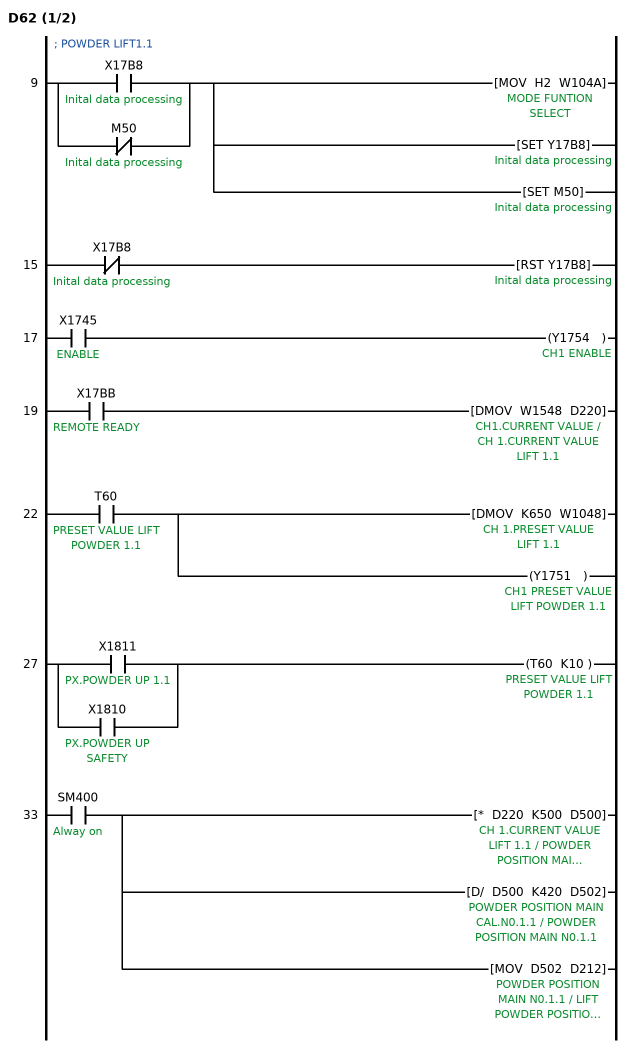
[picture p24: ladder of D62, rungs at steps 9 to 33]
; POWDER LIFT1.1
9     LD      X17B8  ; Inital data processing
      ORI     M50  ; Inital data processing
      MOV     H2 W104A  ; MODE FUNTION SELECT
      SET     Y17B8  ; Inital data processing
      SET     M50  ; Inital data processing
15    LDI     X17B8  ; Inital data processing
      RST     Y17B8  ; Inital data processing
17    LD      X1745  ; ENABLE
      OUT     Y1754  ; CH1 ENABLE
19    LD      X17BB  ; REMOTE READY
      DMOV    W1548 D220  ; CH1.CURRENT VALUE / CH 1.CURRENT VALUE LIFT 1.1
22    LD      T60  ; PRESET VALUE LIFT POWDER 1.1
      DMOV    K650 W1048  ; CH 1.PRESET VALUE LIFT 1.1
      OUT     Y1751  ; CH1 PRESET VALUE LIFT POWDER 1.1
27    LD      X1811  ; PX.POWDER UP 1.1
      OR      X1810  ; PX.POWDER UP SAFETY
      OUT     T60 K10  ; PRESET VALUE LIFT POWDER 1.1
33    LD      SM400  ; Alway on
      *       D220 K500 D500  ; POWDER POSITION MAIN CAL.N0.1.1
      D/      D500 K420 D502  ; POWDER POSITION MAIN N0.1.1
      MOV     D502 D212  ; LIFT POWDER POSITION N0.1.1
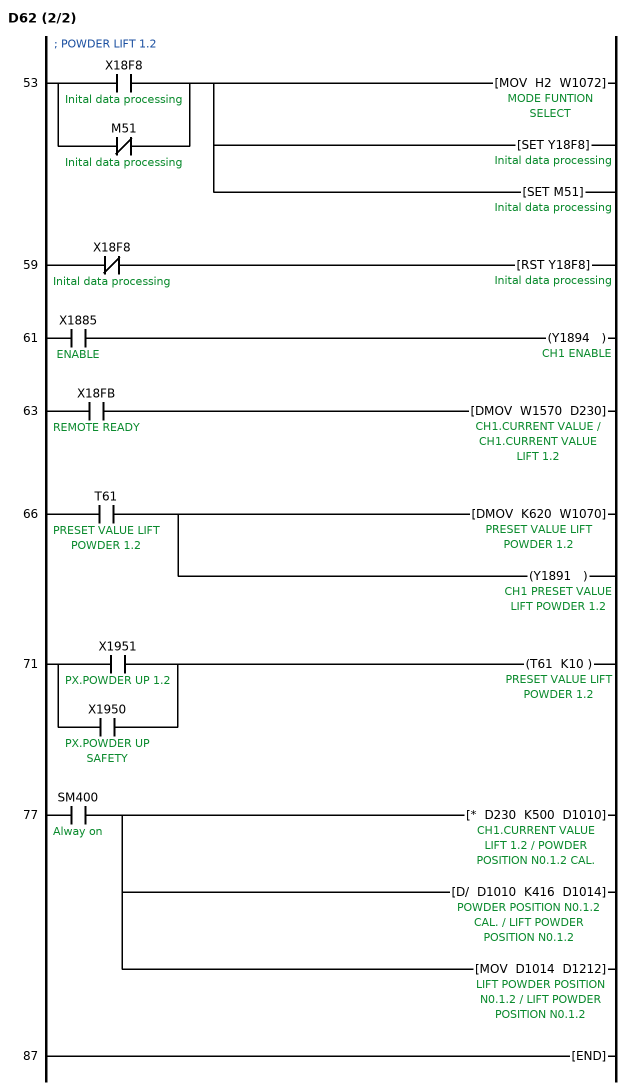
; POWDER LIFT 1.2
53    LD      X18F8  ; Inital data processing
      ORI     M51  ; Inital data processing
      MOV     H2 W1072  ; MODE FUNTION SELECT
      SET     Y18F8  ; Inital data processing
      SET     M51  ; Inital data processing
59    LDI     X18F8  ; Inital data processing
      RST     Y18F8  ; Inital data processing
61    LD      X1885  ; ENABLE
      OUT     Y1894  ; CH1 ENABLE
63    LD      X18FB  ; REMOTE READY
      DMOV    W1570 D230  ; CH1.CURRENT VALUE / CH1.CURRENT VALUE LIFT 1.2
66    LD      T61  ; PRESET VALUE LIFT POWDER 1.2
      DMOV    K620 W1070  ; PRESET VALUE LIFT POWDER 1.2
      OUT     Y1891  ; CH1 PRESET VALUE LIFT POWDER 1.2
71    LD      X1951  ; PX.POWDER UP 1.2
      OR      X1950  ; PX.POWDER UP SAFETY
      OUT     T61 K10  ; PRESET VALUE LIFT POWDER 1.2
77    LD      SM400  ; Alway on
      *       D230 K500 D1010  ; POWDER POSITION N0.1.2 CAL.
      D/      D1010 K416 D1014  ; LIFT POWDER POSITION N0.1.2
      MOV     D1014 D1212  ; LIFT POWDER POSITION N0.1.2
87    END
END_PROGRAM

PROGRAM POWDER1
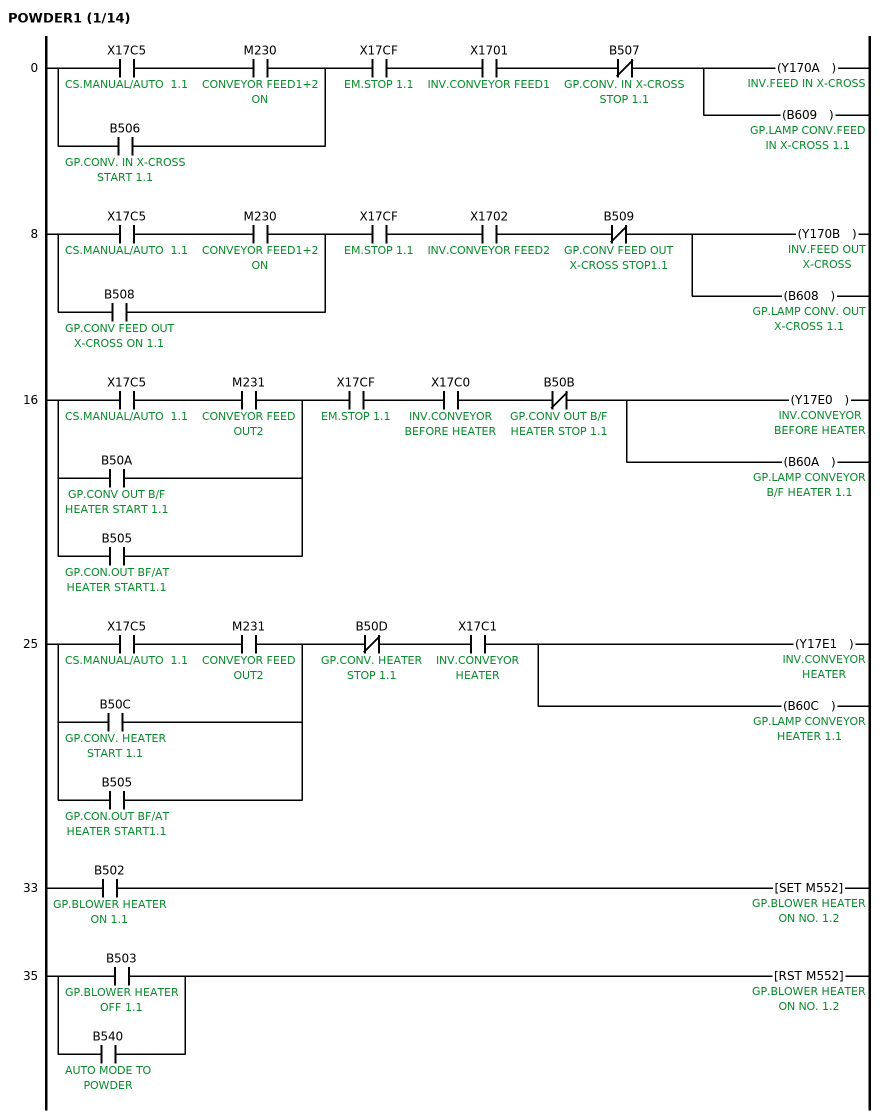
0     LD      X17C5  ; CS.MANUAL/AUTO  1.1
      AND     M230  ; CONVEYOR FEED1+2 ON
      OR      B506  ; GP.CONV. IN X-CROSS START 1.1
      AND     X17CF  ; EM.STOP 1.1
      AND     X1701  ; INV.CONVEYOR FEED1
      ANI     B507  ; GP.CONV. IN X-CROSS STOP 1.1
      OUT     Y170A  ; INV.FEED IN X-CROSS
      OUT     B609  ; GP.LAMP CONV.FEED IN X-CROSS 1.1
8     LD      X17C5  ; CS.MANUAL/AUTO  1.1
      AND     M230  ; CONVEYOR FEED1+2 ON
      OR      B508  ; GP.CONV FEED OUT X-CROSS ON 1.1
      AND     X17CF  ; EM.STOP 1.1
      AND     X1702  ; INV.CONVEYOR FEED2
      ANI     B509  ; GP.CONV FEED OUT X-CROSS STOP1.1
      OUT     Y170B  ; INV.FEED OUT X-CROSS
      OUT     B608  ; GP.LAMP CONV. OUT X-CROSS 1.1
16    LD      X17C5  ; CS.MANUAL/AUTO  1.1
      AND     M231  ; CONVEYOR FEED OUT2
      OR      B50A  ; GP.CONV OUT B/F HEATER START 1.1
      OR      B505  ; GP.CON.OUT BF/AT HEATER START1.1
      AND     X17CF  ; EM.STOP 1.1
      AND     X17C0  ; INV.CONVEYOR BEFORE HEATER
      ANI     B50B  ; GP.CONV OUT B/F HEATER STOP 1.1
      OUT     Y17E0  ; INV.CONVEYOR BEFORE HEATER
      OUT     B60A  ; GP.LAMP CONVEYOR B/F HEATER 1.1
25    LD      X17C5  ; CS.MANUAL/AUTO  1.1
      AND     M231  ; CONVEYOR FEED OUT2
      OR      B50C  ; GP.CONV. HEATER START 1.1
      OR      B505  ; GP.CON.OUT BF/AT HEATER START1.1
      ANI     B50D  ; GP.CONV. HEATER STOP 1.1
      AND     X17C1  ; INV.CONVEYOR HEATER
      OUT     Y17E1  ; INV.CONVEYOR HEATER
      OUT     B60C  ; GP.LAMP CONVEYOR HEATER 1.1
33    LD      B502  ; GP.BLOWER HEATER ON 1.1
      SET     M552  ; GP.BLOWER HEATER ON NO. 1.2
35    LD      B503  ; GP.BLOWER HEATER OFF 1.1
      OR      B540  ; AUTO MODE TO POWDER
      RST     M552  ; GP.BLOWER HEATER ON NO. 1.2
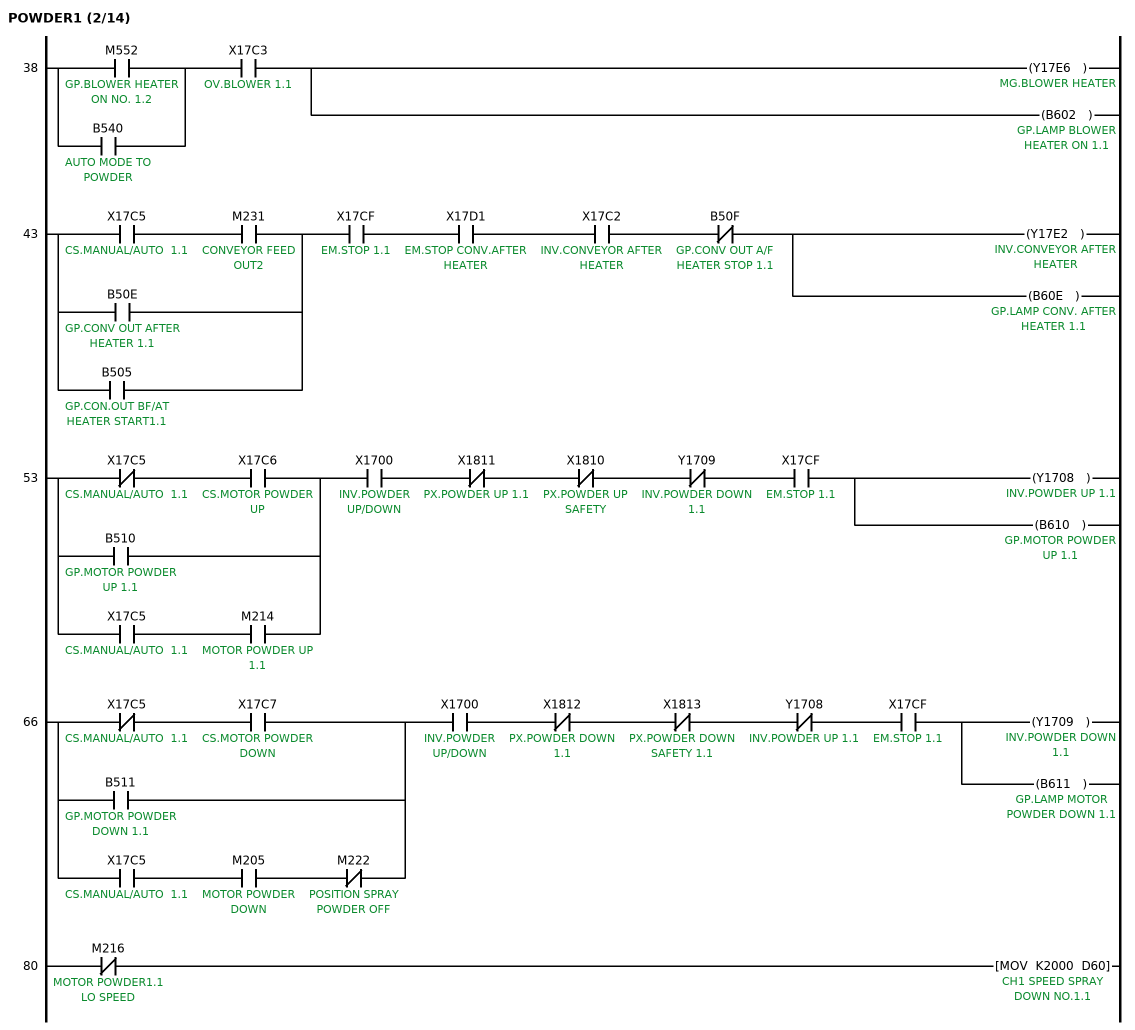
38    LD      M552  ; GP.BLOWER HEATER ON NO. 1.2
      OR      B540  ; AUTO MODE TO POWDER
      AND     X17C3  ; OV.BLOWER 1.1
      OUT     Y17E6  ; MG.BLOWER HEATER
      OUT     B602  ; GP.LAMP BLOWER HEATER ON 1.1
43    LD      X17C5  ; CS.MANUAL/AUTO  1.1
      AND     M231  ; CONVEYOR FEED OUT2
      OR      B50E  ; GP.CONV OUT AFTER HEATER 1.1
      OR      B505  ; GP.CON.OUT BF/AT HEATER START1.1
      AND     X17CF  ; EM.STOP 1.1
      AND     X17D1  ; EM.STOP CONV.AFTER HEATER
      AND     X17C2  ; INV.CONVEYOR AFTER HEATER
      ANI     B50F  ; GP.CONV OUT A/F HEATER STOP 1.1
      OUT     Y17E2  ; INV.CONVEYOR AFTER HEATER
      OUT     B60E  ; GP.LAMP CONV. AFTER HEATER 1.1
53    LDI     X17C5  ; CS.MANUAL/AUTO  1.1
      AND     X17C6  ; CS.MOTOR POWDER UP
      OR      B510  ; GP.MOTOR POWDER UP 1.1
      LD      X17C5  ; CS.MANUAL/AUTO  1.1
      AND     M214  ; MOTOR POWDER UP 1.1
      ORB
      AND     X1700  ; INV.POWDER UP/DOWN
      ANI     X1811  ; PX.POWDER UP 1.1
      ANI     X1810  ; PX.POWDER UP SAFETY
      ANI     Y1709  ; INV.POWDER DOWN 1.1
      AND     X17CF  ; EM.STOP 1.1
      OUT     Y1708  ; INV.POWDER UP 1.1
      OUT     B610  ; GP.MOTOR POWDER UP 1.1
66    LDI     X17C5  ; CS.MANUAL/AUTO  1.1
      AND     X17C7  ; CS.MOTOR POWDER DOWN
      OR      B511  ; GP.MOTOR POWDER DOWN 1.1
      LD      X17C5  ; CS.MANUAL/AUTO  1.1
      AND     M205  ; MOTOR POWDER DOWN
      ANI     M222  ; POSITION SPRAY POWDER OFF
      ORB
      AND     X1700  ; INV.POWDER UP/DOWN
      ANI     X1812  ; PX.POWDER DOWN 1.1
      ANI     X1813  ; PX.POWDER DOWN SAFETY 1.1
      ANI     Y1708  ; INV.POWDER UP 1.1
      AND     X17CF  ; EM.STOP 1.1
      OUT     Y1709  ; INV.POWDER DOWN 1.1
      OUT     B611  ; GP.LAMP MOTOR POWDER DOWN 1.1
80    LDI     M216  ; MOTOR POWDER1.1  LO SPEED
      MOV     K2000 D60  ; CH1 SPEED SPRAY DOWN NO.1.1
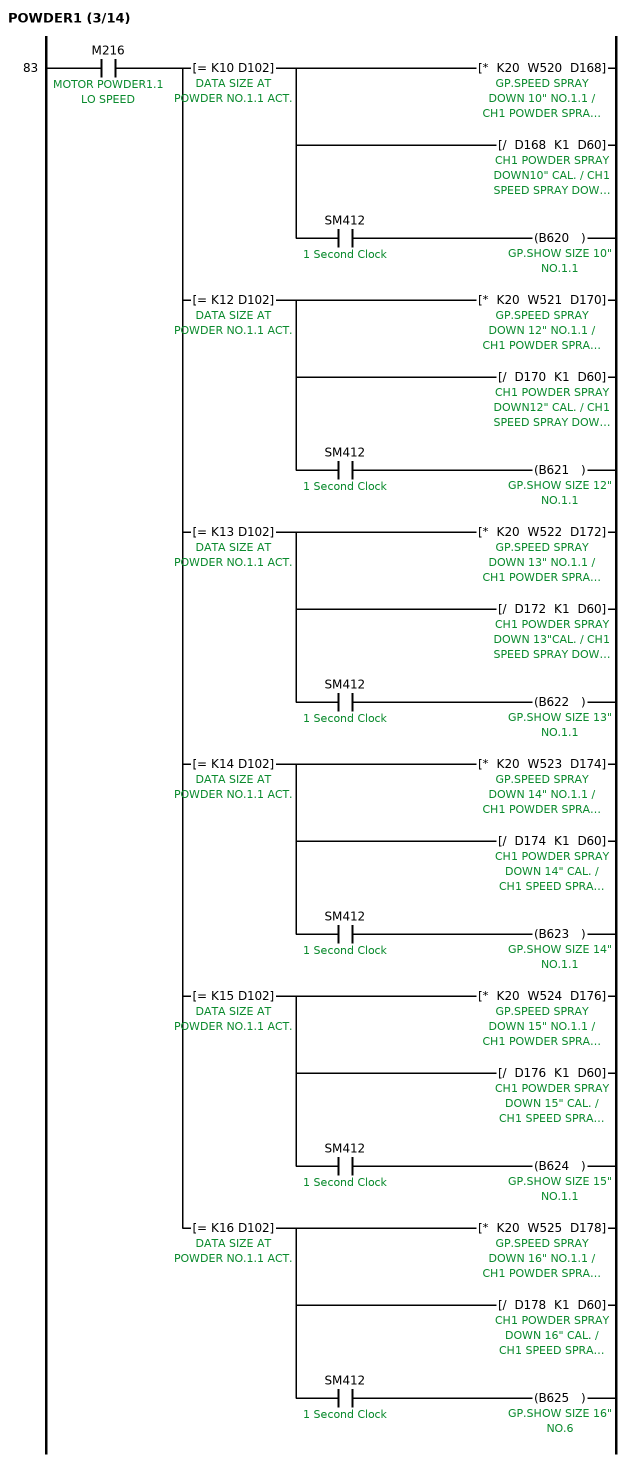
83    LD      M216  ; MOTOR POWDER1.1  LO SPEED
      MPS
      AND=    K10 D102  ; DATA SIZE AT POWDER NO.1.1 ACT.
      *       K20 W520 D168  ; GP.SPEED SPRAY DOWN 10" NO.1.1 / CH1 POWDER SPRAY DOWN10" CAL.
      /       D168 K1 D60
      AND     SM412  ; 1 Second Clock
      OUT     B620  ; GP.SHOW SIZE 10" NO.1.1
      MRD
      AND=    K12 D102  ; DATA SIZE AT POWDER NO.1.1 ACT.
      *       K20 W521 D170  ; GP.SPEED SPRAY DOWN 12" NO.1.1 / CH1 POWDER SPRAY DOWN12" CAL.
      /       D170 K1 D60
      AND     SM412  ; 1 Second Clock
      OUT     B621  ; GP.SHOW SIZE 12" NO.1.1
      MRD
      AND=    K13 D102  ; DATA SIZE AT POWDER NO.1.1 ACT.
      *       K20 W522 D172  ; GP.SPEED SPRAY DOWN 13" NO.1.1 / CH1 POWDER SPRAY DOWN 13"CAL.
      /       D172 K1 D60
      AND     SM412  ; 1 Second Clock
      OUT     B622  ; GP.SHOW SIZE 13" NO.1.1
      MRD
      AND=    K14 D102  ; DATA SIZE AT POWDER NO.1.1 ACT.
      *       K20 W523 D174  ; GP.SPEED SPRAY DOWN 14" NO.1.1 / CH1 POWDER SPRAY DOWN 14" CAL.
      /       D174 K1 D60
      AND     SM412  ; 1 Second Clock
      OUT     B623  ; GP.SHOW SIZE 14" NO.1.1
      MRD
      AND=    K15 D102  ; DATA SIZE AT POWDER NO.1.1 ACT.
      *       K20 W524 D176  ; GP.SPEED SPRAY DOWN 15" NO.1.1 / CH1 POWDER SPRAY DOWN 15" CAL.
      /       D176 K1 D60
      AND     SM412  ; 1 Second Clock
      OUT     B624  ; GP.SHOW SIZE 15" NO.1.1
      MPP
      AND=    K16 D102  ; DATA SIZE AT POWDER NO.1.1 ACT.
      *       K20 W525 D178  ; GP.SPEED SPRAY DOWN 16" NO.1.1 / CH1 POWDER SPRAY DOWN 16" CAL.
      /       D178 K1 D60
      AND     SM412  ; 1 Second Clock
      OUT     B625  ; GP.SHOW SIZE 16" NO.6
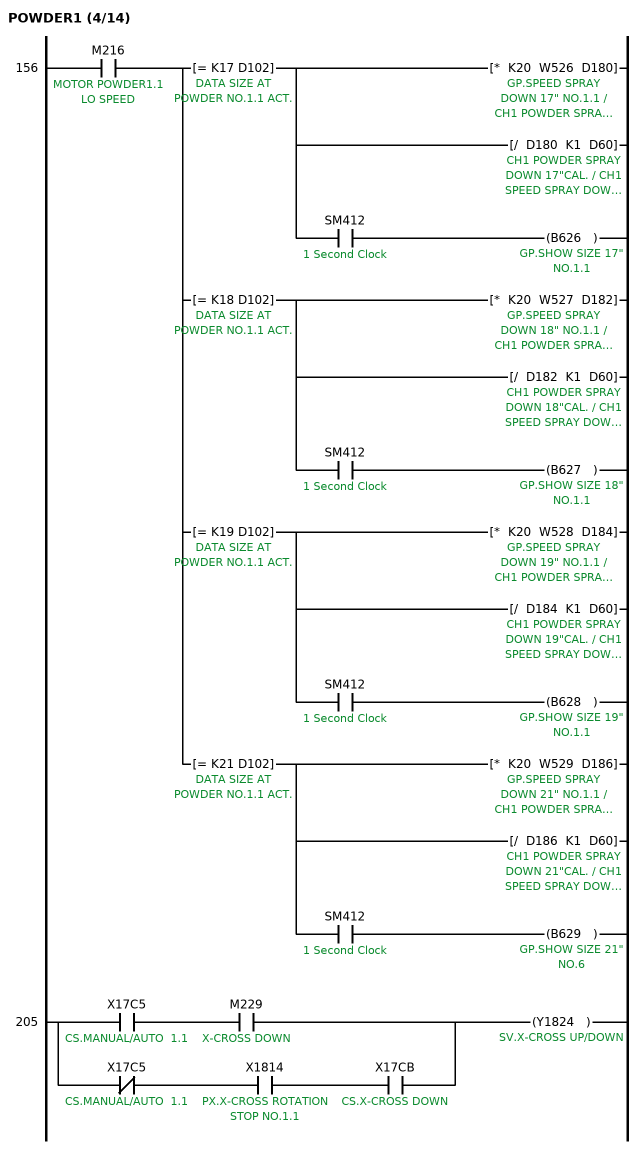
156   LD      M216  ; MOTOR POWDER1.1  LO SPEED
      MPS
      AND=    K17 D102  ; DATA SIZE AT POWDER NO.1.1 ACT.
      *       K20 W526 D180  ; GP.SPEED SPRAY DOWN 17" NO.1.1 / CH1 POWDER SPRAY DOWN 17"CAL.
      /       D180 K1 D60
      AND     SM412  ; 1 Second Clock
      OUT     B626  ; GP.SHOW SIZE 17" NO.1.1
      MRD
      AND=    K18 D102  ; DATA SIZE AT POWDER NO.1.1 ACT.
      *       K20 W527 D182  ; GP.SPEED SPRAY DOWN 18" NO.1.1 / CH1 POWDER SPRAY DOWN 18"CAL.
      /       D182 K1 D60
      AND     SM412  ; 1 Second Clock
      OUT     B627  ; GP.SHOW SIZE 18" NO.1.1
      MRD
      AND=    K19 D102  ; DATA SIZE AT POWDER NO.1.1 ACT.
      *       K20 W528 D184  ; GP.SPEED SPRAY DOWN 19" NO.1.1 / CH1 POWDER SPRAY DOWN 19"CAL.
      /       D184 K1 D60
      AND     SM412  ; 1 Second Clock
      OUT     B628  ; GP.SHOW SIZE 19" NO.1.1
      MPP
      AND=    K21 D102  ; DATA SIZE AT POWDER NO.1.1 ACT.
      *       K20 W529 D186  ; GP.SPEED SPRAY DOWN 21" NO.1.1 / CH1 POWDER SPRAY DOWN 21"CAL.
      /       D186 K1 D60
      AND     SM412  ; 1 Second Clock
      OUT     B629  ; GP.SHOW SIZE 21" NO.6
205   LD      X17C5  ; CS.MANUAL/AUTO  1.1
      AND     M229  ; X-CROSS DOWN
      LDI     X17C5  ; CS.MANUAL/AUTO  1.1
      AND     X1814  ; PX.X-CROSS ROTATION STOP NO.1.1
      AND     X17CB  ; CS.X-CROSS DOWN
      ORB
      OUT     Y1824  ; SV.X-CROSS UP/DOWN
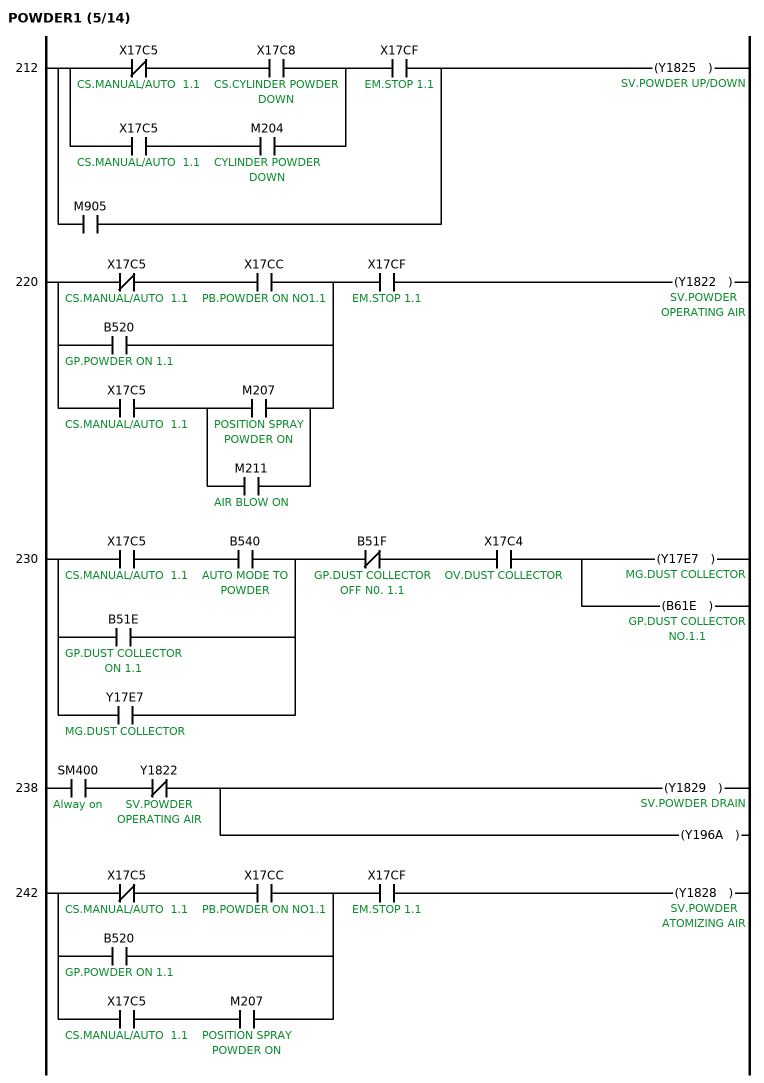
212   LDI     X17C5  ; CS.MANUAL/AUTO  1.1
      AND     X17C8  ; CS.CYLINDER POWDER DOWN
      LD      X17C5  ; CS.MANUAL/AUTO  1.1
      AND     M204  ; CYLINDER POWDER DOWN
      ORB
      AND     X17CF  ; EM.STOP 1.1
      OR      M905
      OUT     Y1825  ; SV.POWDER UP/DOWN
220   LDI     X17C5  ; CS.MANUAL/AUTO  1.1
      AND     X17CC  ; PB.POWDER ON NO1.1
      OR      B520  ; GP.POWDER ON 1.1
      LD      X17C5  ; CS.MANUAL/AUTO  1.1
      LD      M207  ; POSITION SPRAY POWDER ON
      OR      M211  ; AIR BLOW ON
      ANB
      ORB
      AND     X17CF  ; EM.STOP 1.1
      OUT     Y1822  ; SV.POWDER OPERATING AIR
230   LD      X17C5  ; CS.MANUAL/AUTO  1.1
      AND     B540  ; AUTO MODE TO POWDER
      OR      B51E  ; GP.DUST COLLECTOR ON 1.1
      OR      Y17E7  ; MG.DUST COLLECTOR
      ANI     B51F  ; GP.DUST COLLECTOR OFF N0. 1.1
      AND     X17C4  ; OV.DUST COLLECTOR
      OUT     Y17E7  ; MG.DUST COLLECTOR
      OUT     B61E  ; GP.DUST COLLECTOR NO.1.1
238   LD      SM400  ; Alway on
      ANI     Y1822  ; SV.POWDER OPERATING AIR
      OUT     Y1829  ; SV.POWDER DRAIN
      OUT     Y196A
242   LDI     X17C5  ; CS.MANUAL/AUTO  1.1
      AND     X17CC  ; PB.POWDER ON NO1.1
      OR      B520  ; GP.POWDER ON 1.1
      LD      X17C5  ; CS.MANUAL/AUTO  1.1
      AND     M207  ; POSITION SPRAY POWDER ON
      ORB
      AND     X17CF  ; EM.STOP 1.1
      OUT     Y1828  ; SV.POWDER ATOMIZING AIR
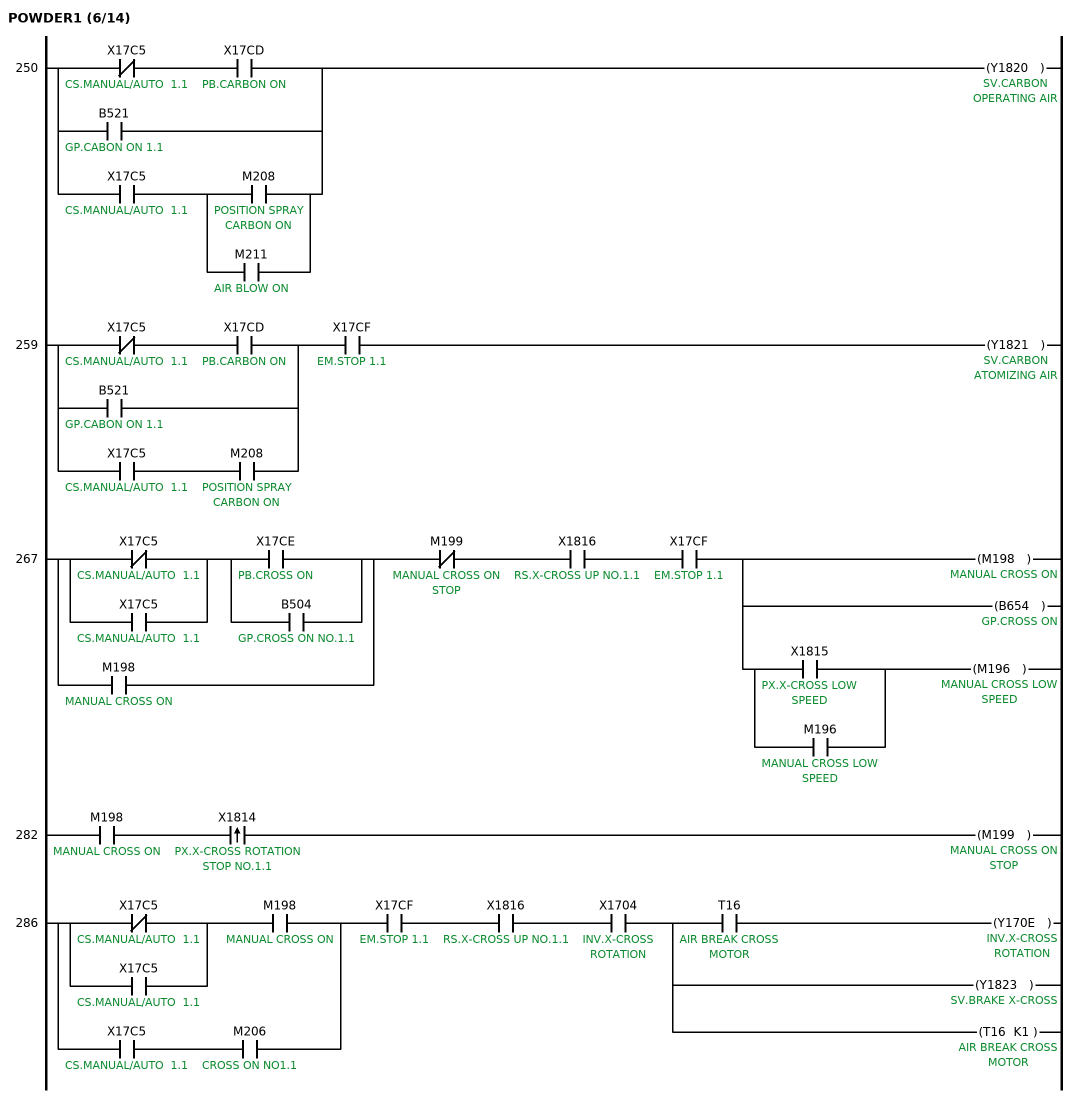
250   LDI     X17C5  ; CS.MANUAL/AUTO  1.1
      AND     X17CD  ; PB.CARBON ON
      OR      B521  ; GP.CABON ON 1.1
      LD      X17C5  ; CS.MANUAL/AUTO  1.1
      LD      M208  ; POSITION SPRAY CARBON ON
      OR      M211  ; AIR BLOW ON
      ANB
      ORB
      OUT     Y1820  ; SV.CARBON OPERATING AIR
259   LDI     X17C5  ; CS.MANUAL/AUTO  1.1
      AND     X17CD  ; PB.CARBON ON
      OR      B521  ; GP.CABON ON 1.1
      LD      X17C5  ; CS.MANUAL/AUTO  1.1
      AND     M208  ; POSITION SPRAY CARBON ON
      ORB
      AND     X17CF  ; EM.STOP 1.1
      OUT     Y1821  ; SV.CARBON ATOMIZING AIR
267   LDI     X17C5  ; CS.MANUAL/AUTO  1.1
      OR      X17C5  ; CS.MANUAL/AUTO  1.1
      LD      X17CE  ; PB.CROSS ON
      OR      B504  ; GP.CROSS ON NO.1.1
      ANB
      OR      M198  ; MANUAL CROSS ON
      ANI     M199  ; MANUAL CROSS ON STOP
      AND     X1816  ; RS.X-CROSS UP NO.1.1
      AND     X17CF  ; EM.STOP 1.1
      OUT     M198  ; MANUAL CROSS ON
      OUT     B654  ; GP.CROSS ON
      LD      X1815  ; PX.X-CROSS LOW SPEED
      OR      M196  ; MANUAL CROSS LOW SPEED
      ANB
      OUT     M196  ; MANUAL CROSS LOW SPEED
282   LD      M198  ; MANUAL CROSS ON
      ANDP    X1814  ; PX.X-CROSS ROTATION STOP NO.1.1
      OUT     M199  ; MANUAL CROSS ON STOP
286   LDI     X17C5  ; CS.MANUAL/AUTO  1.1
      OR      X17C5  ; CS.MANUAL/AUTO  1.1
      AND     M198  ; MANUAL CROSS ON
      LD      X17C5  ; CS.MANUAL/AUTO  1.1
      AND     M206  ; CROSS ON NO1.1
      ORB
      AND     X17CF  ; EM.STOP 1.1
      AND     X1816  ; RS.X-CROSS UP NO.1.1
      AND     X1704  ; INV.X-CROSS ROTATION
      MPS
      AND     T16  ; AIR BREAK CROSS MOTOR
      OUT     Y170E  ; INV.X-CROSS ROTATION
      MPP
      OUT     Y1823  ; SV.BRAKE X-CROSS
      OUT     T16 K1  ; AIR BREAK CROSS MOTOR
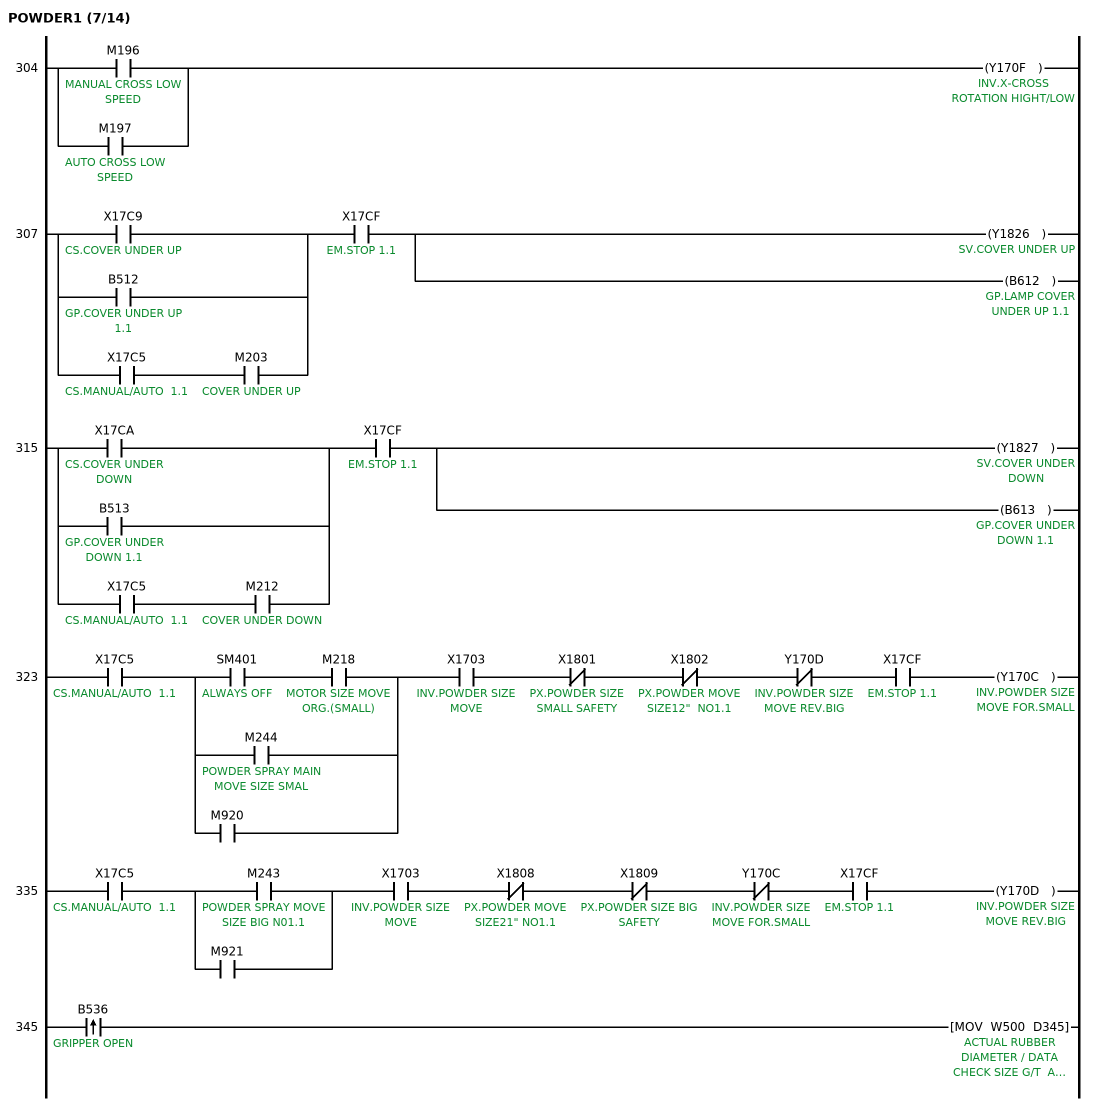
304   LD      M196  ; MANUAL CROSS LOW SPEED
      OR      M197  ; AUTO CROSS LOW SPEED
      OUT     Y170F  ; INV.X-CROSS ROTATION HIGHT/LOW
307   LD      X17C9  ; CS.COVER UNDER UP
      OR      B512  ; GP.COVER UNDER UP 1.1
      LD      X17C5  ; CS.MANUAL/AUTO  1.1
      AND     M203  ; COVER UNDER UP
      ORB
      AND     X17CF  ; EM.STOP 1.1
      OUT     Y1826  ; SV.COVER UNDER UP
      OUT     B612  ; GP.LAMP COVER UNDER UP 1.1
315   LD      X17CA  ; CS.COVER UNDER DOWN
      OR      B513  ; GP.COVER UNDER DOWN 1.1
      LD      X17C5  ; CS.MANUAL/AUTO  1.1
      AND     M212  ; COVER UNDER DOWN
      ORB
      AND     X17CF  ; EM.STOP 1.1
      OUT     Y1827  ; SV.COVER UNDER DOWN
      OUT     B613  ; GP.COVER UNDER DOWN 1.1
323   LD      X17C5  ; CS.MANUAL/AUTO  1.1
      LD      SM401  ; ALWAYS OFF
      AND     M218  ; MOTOR SIZE MOVE ORG.(SMALL)
      OR      M244  ; POWDER SPRAY MAIN MOVE SIZE SMAL
      OR      M920
      ANB
      AND     X1703  ; INV.POWDER SIZE MOVE
      ANI     X1801  ; PX.POWDER SIZE SMALL SAFETY
      ANI     X1802  ; PX.POWDER MOVE  SIZE12"  NO1.1
      ANI     Y170D  ; INV.POWDER SIZE MOVE REV.BIG
      AND     X17CF  ; EM.STOP 1.1
      OUT     Y170C  ; INV.POWDER SIZE MOVE FOR.SMALL
335   LD      X17C5  ; CS.MANUAL/AUTO  1.1
      LD      M243  ; POWDER SPRAY MOVE SIZE BIG N01.1
      OR      M921
      ANB
      AND     X1703  ; INV.POWDER SIZE MOVE
      ANI     X1808  ; PX.POWDER MOVE SIZE21" NO1.1
      ANI     X1809  ; PX.POWDER SIZE BIG SAFETY
      ANI     Y170C  ; INV.POWDER SIZE MOVE FOR.SMALL
      AND     X17CF  ; EM.STOP 1.1
      OUT     Y170D  ; INV.POWDER SIZE MOVE REV.BIG
345   LDP     B536  ; GRIPPER OPEN
      MOV     W500 D345  ; ACTUAL RUBBER DIAMETER / DATA CHECK SIZE G/T  AT ROBOT
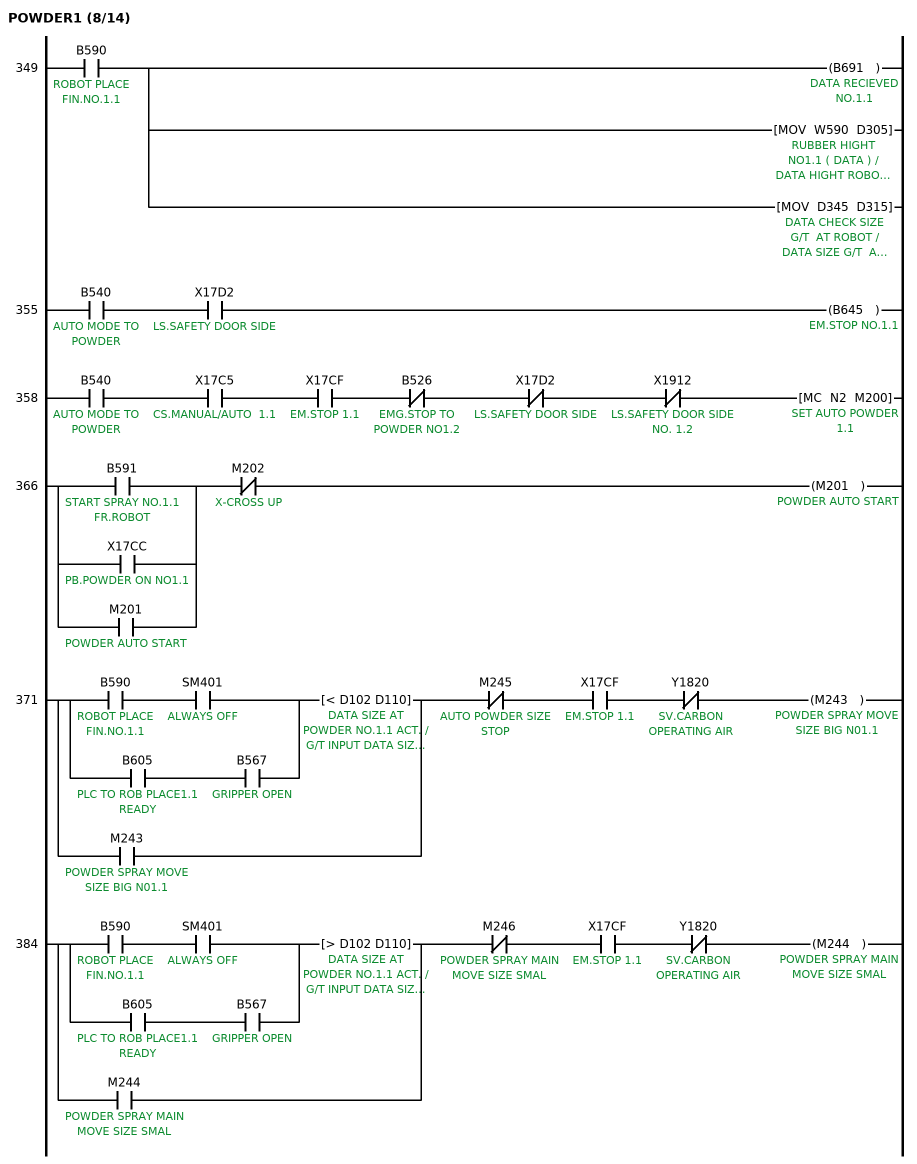
349   LD      B590  ; ROBOT PLACE FIN.NO.1.1
      OUT     B691  ; DATA RECIEVED NO.1.1
      MOV     W590 D305  ; RUBBER HIGHT NO1.1 ( DATA ) / DATA HIGHT ROBOT TO N0.1.1
      MOV     D345 D315  ; DATA SIZE G/T  AT ROBOT NO.1.1
355   LD      B540  ; AUTO MODE TO POWDER
      AND     X17D2  ; LS.SAFETY DOOR SIDE
      OUT     B645  ; EM.STOP NO.1.1
358   LD      B540  ; AUTO MODE TO POWDER
      AND     X17C5  ; CS.MANUAL/AUTO  1.1
      AND     X17CF  ; EM.STOP 1.1
      ANI     B526  ; EMG.STOP TO POWDER NO1.2
      ANI     X17D2  ; LS.SAFETY DOOR SIDE
      ANI     X1912  ; LS.SAFETY DOOR SIDE NO. 1.2
      MC      N2 M200  ; SET AUTO POWDER 1.1
366   LD      B591  ; START SPRAY NO.1.1 FR.ROBOT
      OR      X17CC  ; PB.POWDER ON NO1.1
      OR      M201  ; POWDER AUTO START
      ANI     M202  ; X-CROSS UP
      OUT     M201  ; POWDER AUTO START
371   LD      B590  ; ROBOT PLACE FIN.NO.1.1
      AND     SM401  ; ALWAYS OFF
      LD      B605  ; PLC TO ROB PLACE1.1 READY
      AND     B567  ; GRIPPER OPEN
      ORB
      AND<    D102 D110  ; DATA SIZE AT POWDER NO.1.1 ACT. / G/T INPUT DATA SIZE AT ROBOT
      OR      M243  ; POWDER SPRAY MOVE SIZE BIG N01.1
      ANI     M245  ; AUTO POWDER SIZE STOP
      AND     X17CF  ; EM.STOP 1.1
      ANI     Y1820  ; SV.CARBON OPERATING AIR
      OUT     M243  ; POWDER SPRAY MOVE SIZE BIG N01.1
384   LD      B590  ; ROBOT PLACE FIN.NO.1.1
      AND     SM401  ; ALWAYS OFF
      LD      B605  ; PLC TO ROB PLACE1.1 READY
      AND     B567  ; GRIPPER OPEN
      ORB
      AND>    D102 D110  ; DATA SIZE AT POWDER NO.1.1 ACT. / G/T INPUT DATA SIZE AT ROBOT
      OR      M244  ; POWDER SPRAY MAIN MOVE SIZE SMAL
      ANI     M246  ; POWDER SPRAY MAIN MOVE SIZE SMAL
      AND     X17CF  ; EM.STOP 1.1
      ANI     Y1820  ; SV.CARBON OPERATING AIR
      OUT     M244  ; POWDER SPRAY MAIN MOVE SIZE SMAL
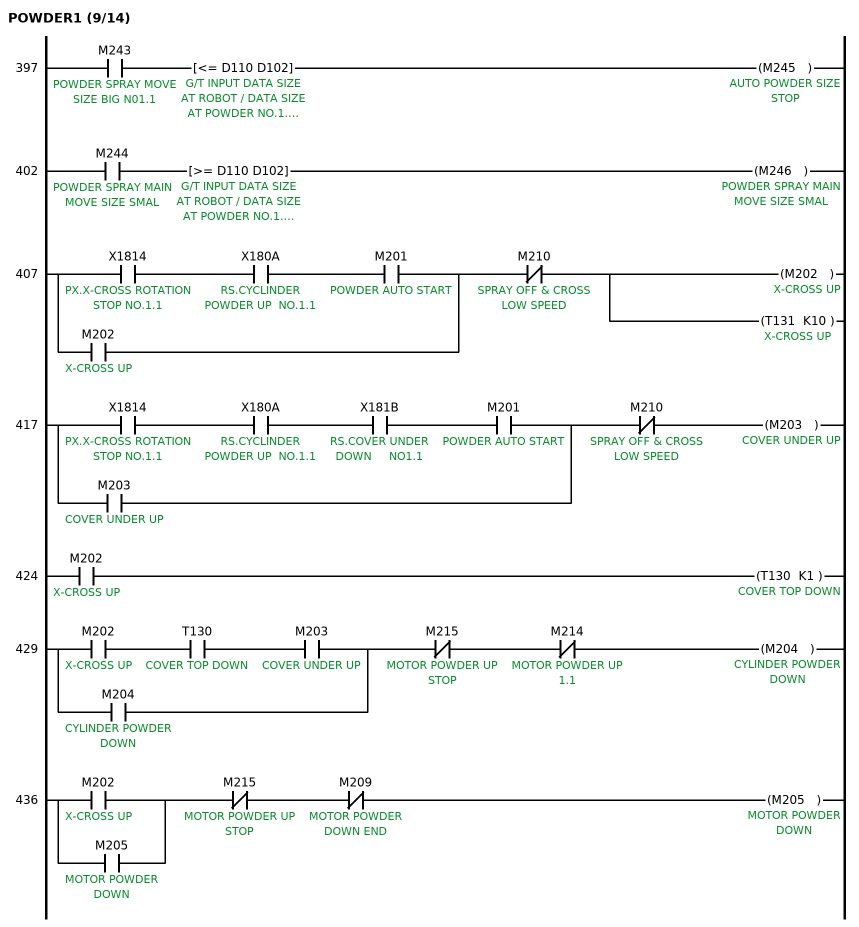
397   LD      M243  ; POWDER SPRAY MOVE SIZE BIG N01.1
      AND<=   D110 D102  ; G/T INPUT DATA SIZE AT ROBOT / DATA SIZE AT POWDER NO.1.1 ACT.
      OUT     M245  ; AUTO POWDER SIZE STOP
402   LD      M244  ; POWDER SPRAY MAIN MOVE SIZE SMAL
      AND>=   D110 D102  ; G/T INPUT DATA SIZE AT ROBOT / DATA SIZE AT POWDER NO.1.1 ACT.
      OUT     M246  ; POWDER SPRAY MAIN MOVE SIZE SMAL
407   LD      X1814  ; PX.X-CROSS ROTATION STOP NO.1.1
      AND     X180A  ; RS.CYCLINDER POWDER UP  NO.1.1
      AND     M201  ; POWDER AUTO START
      OR      M202  ; X-CROSS UP
      ANI     M210  ; SPRAY OFF & CROSS LOW SPEED
      OUT     M202  ; X-CROSS UP
      OUT     T131 K10  ; X-CROSS UP
417   LD      X1814  ; PX.X-CROSS ROTATION STOP NO.1.1
      AND     X180A  ; RS.CYCLINDER POWDER UP  NO.1.1
      AND     X181B  ; RS.COVER UNDER DOWN     NO1.1
      AND     M201  ; POWDER AUTO START
      OR      M203  ; COVER UNDER UP
      ANI     M210  ; SPRAY OFF & CROSS LOW SPEED
      OUT     M203  ; COVER UNDER UP
424   LD      M202  ; X-CROSS UP
      OUT     T130 K1  ; COVER TOP DOWN
429   LD      M202  ; X-CROSS UP
      AND     T130  ; COVER TOP DOWN
      AND     M203  ; COVER UNDER UP
      OR      M204  ; CYLINDER POWDER DOWN
      ANI     M215  ; MOTOR POWDER UP STOP
      ANI     M214  ; MOTOR POWDER UP 1.1
      OUT     M204  ; CYLINDER POWDER DOWN
436   LD      M202  ; X-CROSS UP
      OR      M205  ; MOTOR POWDER DOWN
      ANI     M215  ; MOTOR POWDER UP STOP
      ANI     M209  ; MOTOR POWDER DOWN END
      OUT     M205  ; MOTOR POWDER DOWN
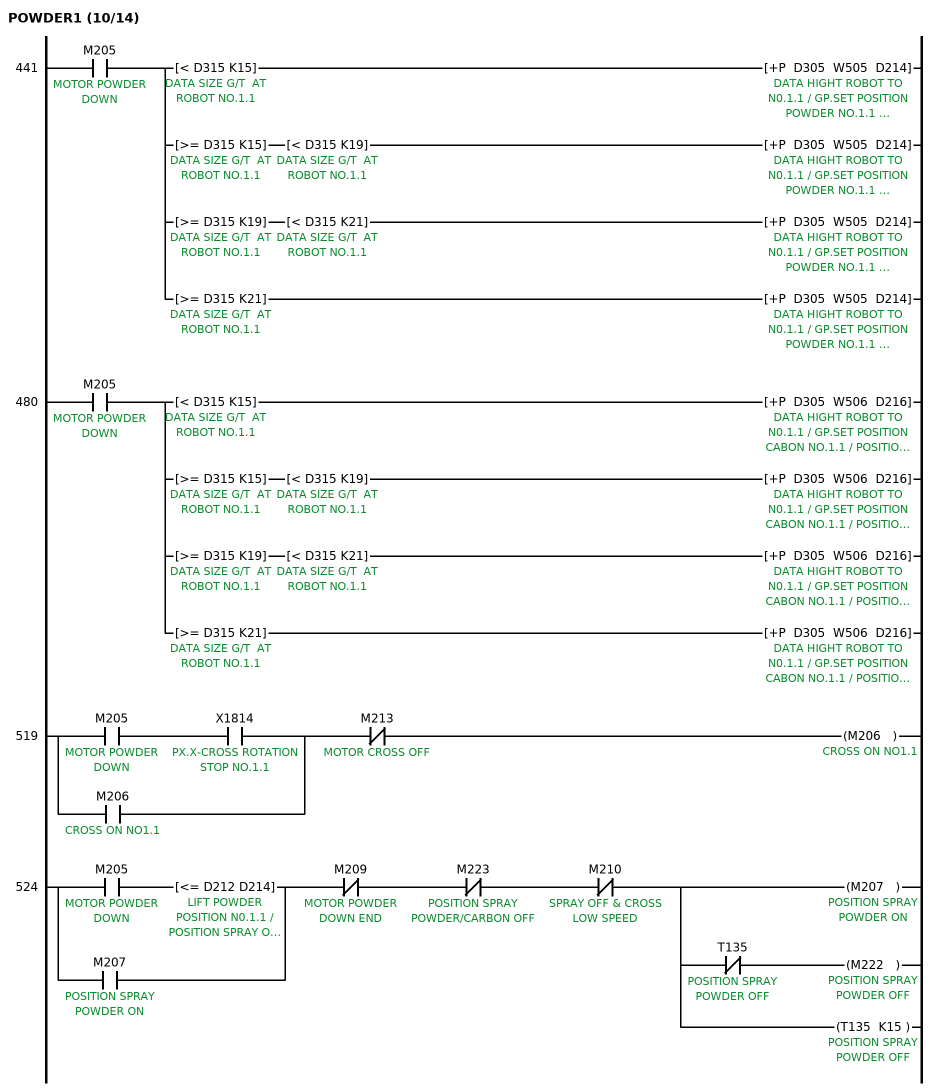
441   LD      M205  ; MOTOR POWDER DOWN
      MPS
      AND<    D315 K15  ; DATA SIZE G/T  AT ROBOT NO.1.1
      +P      D305 W505 D214  ; GP.SET POSITION POWDER NO.1.1 / POSITION SPRAY ON 1.1
      MRD
      AND>=   D315 K15  ; DATA SIZE G/T  AT ROBOT NO.1.1
      AND<    D315 K19  ; DATA SIZE G/T  AT ROBOT NO.1.1
      +P      D305 W505 D214
      MRD
      AND>=   D315 K19  ; DATA SIZE G/T  AT ROBOT NO.1.1
      AND<    D315 K21  ; DATA SIZE G/T  AT ROBOT NO.1.1
      +P      D305 W505 D214
      MPP
      AND>=   D315 K21  ; DATA SIZE G/T  AT ROBOT NO.1.1
      +P      D305 W505 D214
480   LD      M205  ; MOTOR POWDER DOWN
      MPS
      AND<    D315 K15  ; DATA SIZE G/T  AT ROBOT NO.1.1
      +P      D305 W506 D216  ; GP.SET POSITION CABON NO.1.1 / POSITION CARBON ON 1.1
      MRD
      AND>=   D315 K15  ; DATA SIZE G/T  AT ROBOT NO.1.1
      AND<    D315 K19  ; DATA SIZE G/T  AT ROBOT NO.1.1
      +P      D305 W506 D216
      MRD
      AND>=   D315 K19  ; DATA SIZE G/T  AT ROBOT NO.1.1
      AND<    D315 K21  ; DATA SIZE G/T  AT ROBOT NO.1.1
      +P      D305 W506 D216
      MPP
      AND>=   D315 K21  ; DATA SIZE G/T  AT ROBOT NO.1.1
      +P      D305 W506 D216
519   LD      M205  ; MOTOR POWDER DOWN
      AND     X1814  ; PX.X-CROSS ROTATION STOP NO.1.1
      OR      M206  ; CROSS ON NO1.1
      ANI     M213  ; MOTOR CROSS OFF
      OUT     M206  ; CROSS ON NO1.1
524   LD      M205  ; MOTOR POWDER DOWN
      AND<=   D212 D214  ; LIFT POWDER POSITION N0.1.1 / POSITION SPRAY ON 1.1
      OR      M207  ; POSITION SPRAY POWDER ON
      ANI     M209  ; MOTOR POWDER DOWN END
      ANI     M223  ; POSITION SPRAY POWDER/CARBON OFF
      ANI     M210  ; SPRAY OFF & CROSS LOW SPEED
      OUT     M207  ; POSITION SPRAY POWDER ON
      MPS
      ANI     T135  ; POSITION SPRAY POWDER OFF
      OUT     M222  ; POSITION SPRAY POWDER OFF
      MPP
      OUT     T135 K15  ; POSITION SPRAY POWDER OFF
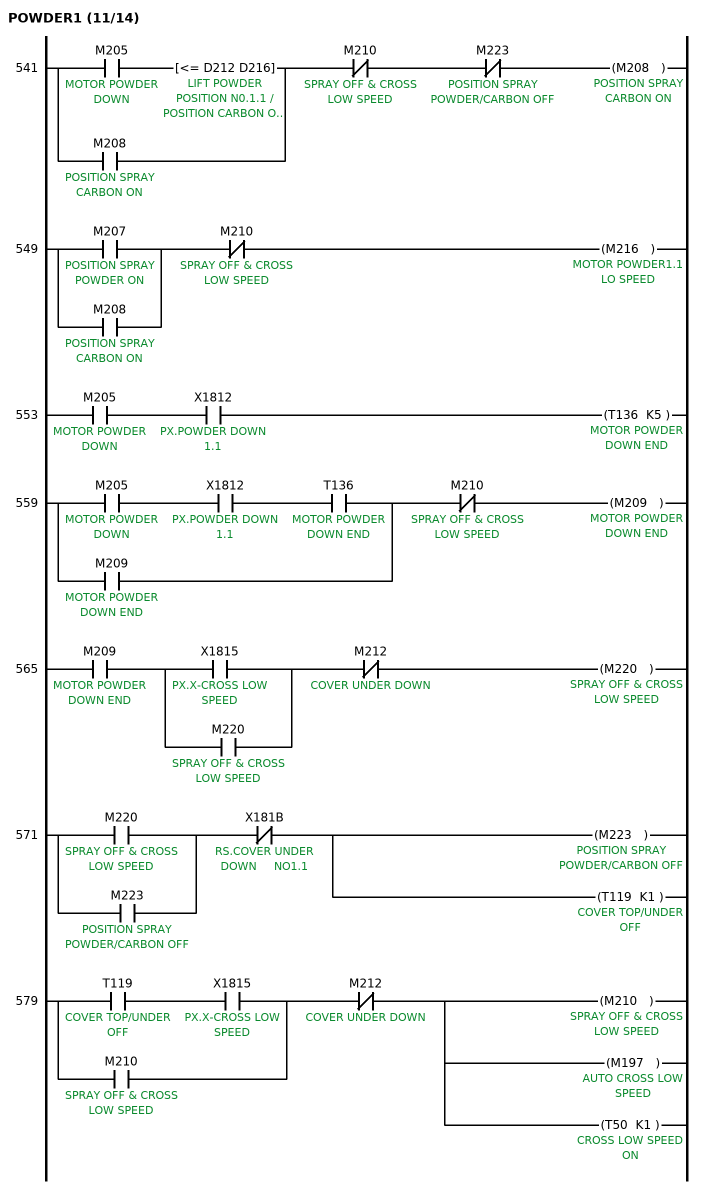
541   LD      M205  ; MOTOR POWDER DOWN
      AND<=   D212 D216  ; LIFT POWDER POSITION N0.1.1 / POSITION CARBON ON 1.1
      OR      M208  ; POSITION SPRAY CARBON ON
      ANI     M210  ; SPRAY OFF & CROSS LOW SPEED
      ANI     M223  ; POSITION SPRAY POWDER/CARBON OFF
      OUT     M208  ; POSITION SPRAY CARBON ON
549   LD      M207  ; POSITION SPRAY POWDER ON
      OR      M208  ; POSITION SPRAY CARBON ON
      ANI     M210  ; SPRAY OFF & CROSS LOW SPEED
      OUT     M216  ; MOTOR POWDER1.1  LO SPEED
553   LD      M205  ; MOTOR POWDER DOWN
      AND     X1812  ; PX.POWDER DOWN 1.1
      OUT     T136 K5  ; MOTOR POWDER DOWN END
559   LD      M205  ; MOTOR POWDER DOWN
      AND     X1812  ; PX.POWDER DOWN 1.1
      AND     T136  ; MOTOR POWDER DOWN END
      OR      M209  ; MOTOR POWDER DOWN END
      ANI     M210  ; SPRAY OFF & CROSS LOW SPEED
      OUT     M209  ; MOTOR POWDER DOWN END
565   LD      M209  ; MOTOR POWDER DOWN END
      LD      X1815  ; PX.X-CROSS LOW SPEED
      OR      M220  ; SPRAY OFF & CROSS LOW SPEED
      ANB
      ANI     M212  ; COVER UNDER DOWN
      OUT     M220  ; SPRAY OFF & CROSS LOW SPEED
571   LD      M220  ; SPRAY OFF & CROSS LOW SPEED
      OR      M223  ; POSITION SPRAY POWDER/CARBON OFF
      ANI     X181B  ; RS.COVER UNDER DOWN     NO1.1
      OUT     M223  ; POSITION SPRAY POWDER/CARBON OFF
      OUT     T119 K1  ; COVER TOP/UNDER OFF
579   LD      T119  ; COVER TOP/UNDER OFF
      AND     X1815  ; PX.X-CROSS LOW SPEED
      OR      M210  ; SPRAY OFF & CROSS LOW SPEED
      ANI     M212  ; COVER UNDER DOWN
      OUT     M210  ; SPRAY OFF & CROSS LOW SPEED
      OUT     M197  ; AUTO CROSS LOW SPEED
      OUT     T50 K1  ; CROSS LOW SPEED ON
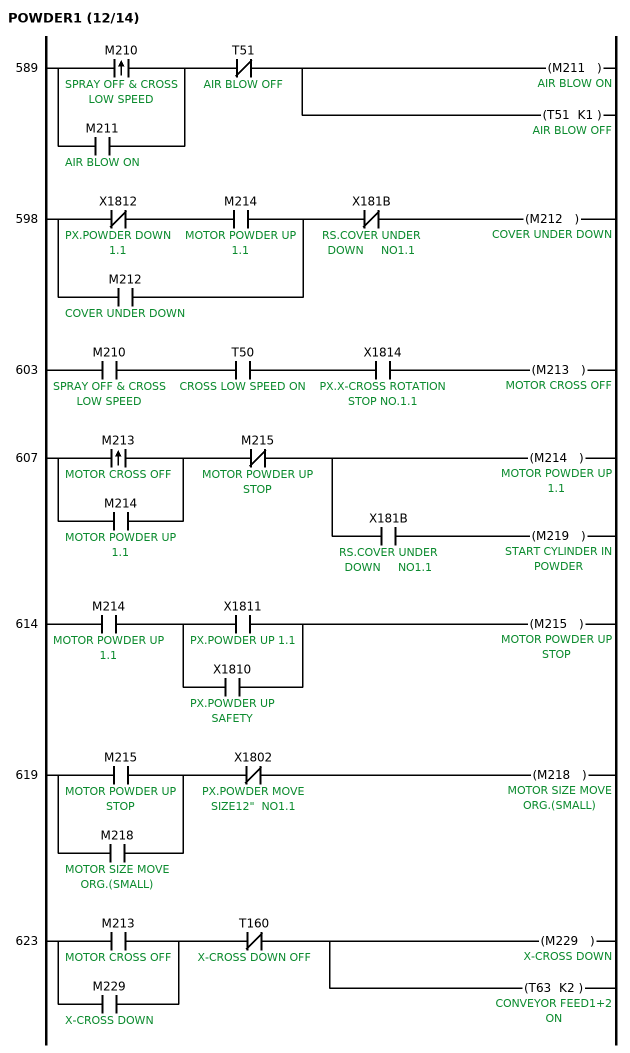
589   LDP     M210  ; SPRAY OFF & CROSS LOW SPEED
      OR      M211  ; AIR BLOW ON
      ANI     T51  ; AIR BLOW OFF
      OUT     M211  ; AIR BLOW ON
      OUT     T51 K1  ; AIR BLOW OFF
598   LDI     X1812  ; PX.POWDER DOWN 1.1
      AND     M214  ; MOTOR POWDER UP 1.1
      OR      M212  ; COVER UNDER DOWN
      ANI     X181B  ; RS.COVER UNDER DOWN     NO1.1
      OUT     M212  ; COVER UNDER DOWN
603   LD      M210  ; SPRAY OFF & CROSS LOW SPEED
      AND     T50  ; CROSS LOW SPEED ON
      AND     X1814  ; PX.X-CROSS ROTATION STOP NO.1.1
      OUT     M213  ; MOTOR CROSS OFF
607   LDP     M213  ; MOTOR CROSS OFF
      OR      M214  ; MOTOR POWDER UP 1.1
      ANI     M215  ; MOTOR POWDER UP STOP
      OUT     M214  ; MOTOR POWDER UP 1.1
      AND     X181B  ; RS.COVER UNDER DOWN     NO1.1
      OUT     M219  ; START CYLINDER IN POWDER
614   LD      M214  ; MOTOR POWDER UP 1.1
      LD      X1811  ; PX.POWDER UP 1.1
      OR      X1810  ; PX.POWDER UP SAFETY
      ANB
      OUT     M215  ; MOTOR POWDER UP STOP
619   LD      M215  ; MOTOR POWDER UP STOP
      OR      M218  ; MOTOR SIZE MOVE ORG.(SMALL)
      ANI     X1802  ; PX.POWDER MOVE  SIZE12"  NO1.1
      OUT     M218  ; MOTOR SIZE MOVE ORG.(SMALL)
623   LD      M213  ; MOTOR CROSS OFF
      OR      M229  ; X-CROSS DOWN
      ANI     T160  ; X-CROSS DOWN OFF
      OUT     M229  ; X-CROSS DOWN
      OUT     T63 K2  ; CONVEYOR FEED1+2 ON
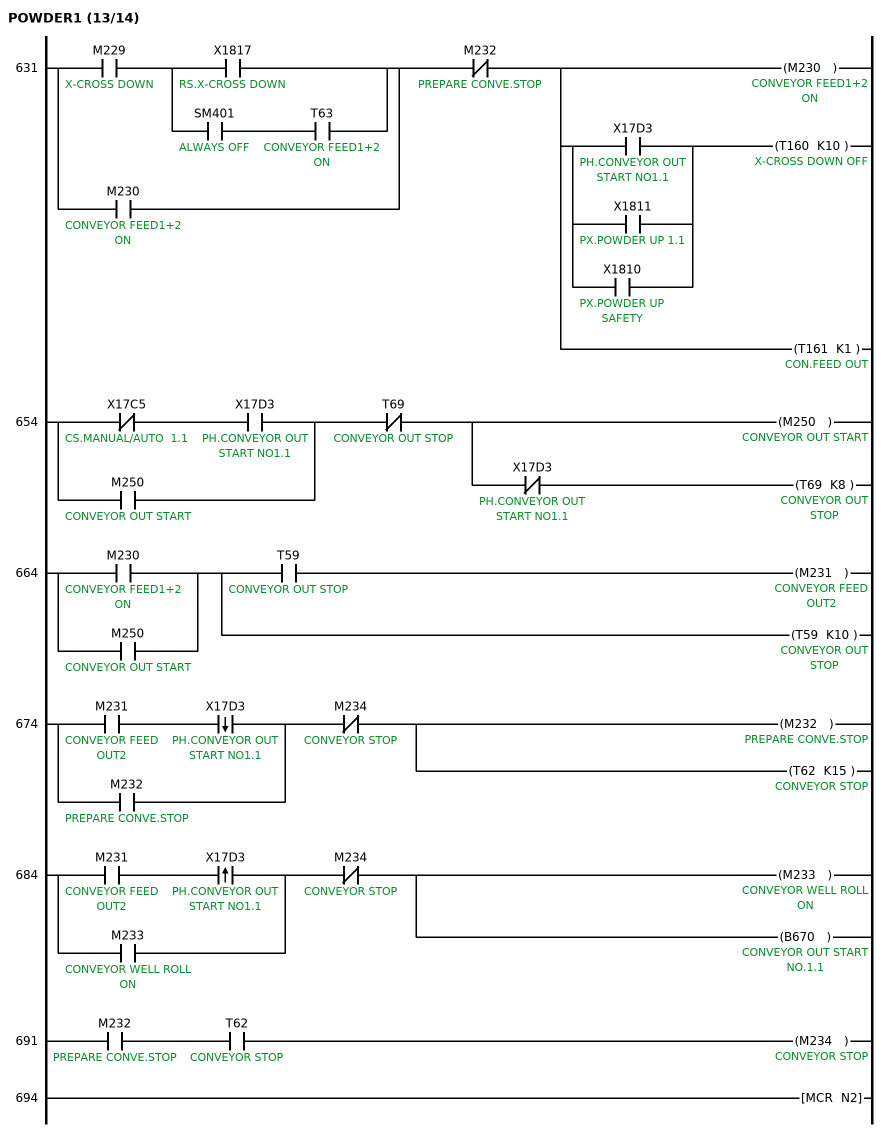
631   LD      M229  ; X-CROSS DOWN
      LD      X1817  ; RS.X-CROSS DOWN
      LD      SM401  ; ALWAYS OFF
      AND     T63  ; CONVEYOR FEED1+2 ON
      ORB
      ANB
      OR      M230  ; CONVEYOR FEED1+2 ON
      ANI     M232  ; PREPARE CONVE.STOP
      OUT     M230  ; CONVEYOR FEED1+2 ON
      MPS
      LD      X17D3  ; PH.CONVEYOR OUT START NO1.1
      OR      X1811  ; PX.POWDER UP 1.1
      OR      X1810  ; PX.POWDER UP SAFETY
      ANB
      OUT     T160 K10  ; X-CROSS DOWN OFF
      MPP
      OUT     T161 K1  ; CON.FEED OUT
654   LDI     X17C5  ; CS.MANUAL/AUTO  1.1
      AND     X17D3  ; PH.CONVEYOR OUT START NO1.1
      OR      M250  ; CONVEYOR OUT START
      ANI     T69  ; CONVEYOR OUT STOP
      OUT     M250  ; CONVEYOR OUT START
      ANI     X17D3  ; PH.CONVEYOR OUT START NO1.1
      OUT     T69 K8  ; CONVEYOR OUT STOP
664   LD      M230  ; CONVEYOR FEED1+2 ON
      OR      M250  ; CONVEYOR OUT START
      MPS
      AND     T59  ; CONVEYOR OUT STOP
      OUT     M231  ; CONVEYOR FEED OUT2
      MPP
      OUT     T59 K10  ; CONVEYOR OUT STOP
674   LD      M231  ; CONVEYOR FEED OUT2
      ANDF    X17D3  ; PH.CONVEYOR OUT START NO1.1
      OR      M232  ; PREPARE CONVE.STOP
      ANI     M234  ; CONVEYOR STOP
      OUT     M232  ; PREPARE CONVE.STOP
      OUT     T62 K15  ; CONVEYOR STOP
684   LD      M231  ; CONVEYOR FEED OUT2
      ANDP    X17D3  ; PH.CONVEYOR OUT START NO1.1
      OR      M233  ; CONVEYOR WELL ROLL ON
      ANI     M234  ; CONVEYOR STOP
      OUT     M233  ; CONVEYOR WELL ROLL ON
      OUT     B670  ; CONVEYOR OUT START NO.1.1
691   LD      M232  ; PREPARE CONVE.STOP
      AND     T62  ; CONVEYOR STOP
      OUT     M234  ; CONVEYOR STOP
694   MCR     N2
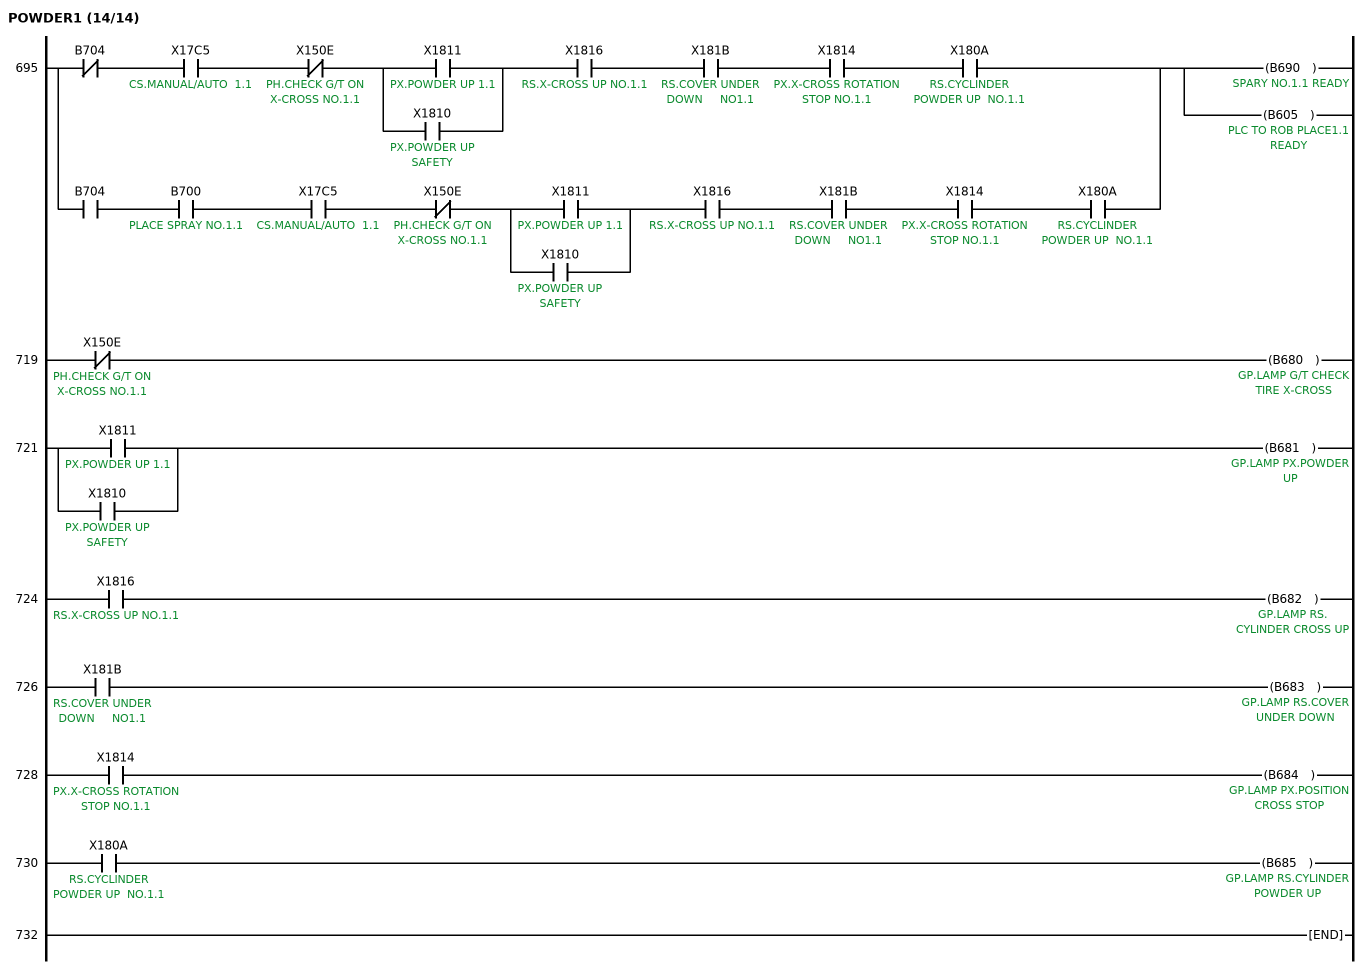
695   LDI     B704
      AND     X17C5  ; CS.MANUAL/AUTO  1.1
      ANI     X150E  ; PH.CHECK G/T ON X-CROSS NO.1.1
      LD      X1811  ; PX.POWDER UP 1.1
      OR      X1810  ; PX.POWDER UP SAFETY
      ANB
      AND     X1816  ; RS.X-CROSS UP NO.1.1
      AND     X181B  ; RS.COVER UNDER DOWN     NO1.1
      AND     X1814  ; PX.X-CROSS ROTATION STOP NO.1.1
      AND     X180A  ; RS.CYCLINDER POWDER UP  NO.1.1
      LD      B704
      AND     B700  ; PLACE SPRAY NO.1.1
      AND     X17C5  ; CS.MANUAL/AUTO  1.1
      ANI     X150E  ; PH.CHECK G/T ON X-CROSS NO.1.1
      LD      X1811  ; PX.POWDER UP 1.1
      OR      X1810  ; PX.POWDER UP SAFETY
      ANB
      AND     X1816  ; RS.X-CROSS UP NO.1.1
      AND     X181B  ; RS.COVER UNDER DOWN     NO1.1
      AND     X1814  ; PX.X-CROSS ROTATION STOP NO.1.1
      AND     X180A  ; RS.CYCLINDER POWDER UP  NO.1.1
      ORB
      OUT     B690  ; SPARY NO.1.1 READY
      OUT     B605  ; PLC TO ROB PLACE1.1 READY
719   LDI     X150E  ; PH.CHECK G/T ON X-CROSS NO.1.1
      OUT     B680  ; GP.LAMP G/T CHECK TIRE X-CROSS
721   LD      X1811  ; PX.POWDER UP 1.1
      OR      X1810  ; PX.POWDER UP SAFETY
      OUT     B681  ; GP.LAMP PX.POWDER UP
724   LD      X1816  ; RS.X-CROSS UP NO.1.1
      OUT     B682  ; GP.LAMP RS. CYLINDER CROSS UP
726   LD      X181B  ; RS.COVER UNDER DOWN     NO1.1
      OUT     B683  ; GP.LAMP RS.COVER UNDER DOWN
728   LD      X1814  ; PX.X-CROSS ROTATION STOP NO.1.1
      OUT     B684  ; GP.LAMP PX.POSITION CROSS STOP
730   LD      X180A  ; RS.CYCLINDER POWDER UP  NO.1.1
      OUT     B685  ; GP.LAMP RS.CYLINDER POWDER UP
732   END
END_PROGRAM

PROGRAM POWDER2
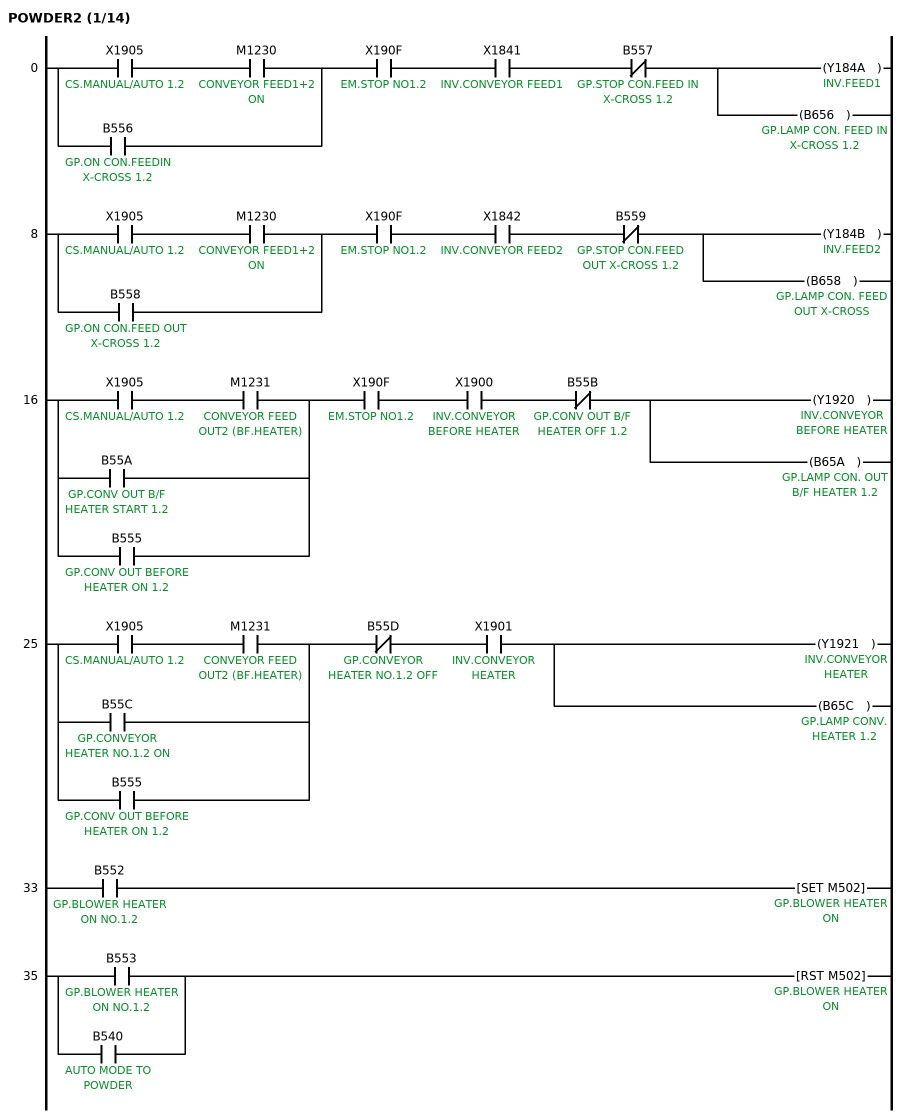
0     LD      X1905  ; CS.MANUAL/AUTO 1.2
      AND     M1230  ; CONVEYOR FEED1+2 ON
      OR      B556  ; GP.ON CON.FEEDIN X-CROSS 1.2
      AND     X190F  ; EM.STOP NO1.2
      AND     X1841  ; INV.CONVEYOR FEED1
      ANI     B557  ; GP.STOP CON.FEED IN X-CROSS 1.2
      OUT     Y184A  ; INV.FEED1
      OUT     B656  ; GP.LAMP CON. FEED IN X-CROSS 1.2
8     LD      X1905  ; CS.MANUAL/AUTO 1.2
      AND     M1230  ; CONVEYOR FEED1+2 ON
      OR      B558  ; GP.ON CON.FEED OUT X-CROSS 1.2
      AND     X190F  ; EM.STOP NO1.2
      AND     X1842  ; INV.CONVEYOR FEED2
      ANI     B559  ; GP.STOP CON.FEED OUT X-CROSS 1.2
      OUT     Y184B  ; INV.FEED2
      OUT     B658  ; GP.LAMP CON. FEED OUT X-CROSS
16    LD      X1905  ; CS.MANUAL/AUTO 1.2
      AND     M1231  ; CONVEYOR FEED OUT2 (BF.HEATER)
      OR      B55A  ; GP.CONV OUT B/F HEATER START 1.2
      OR      B555  ; GP.CONV OUT BEFORE HEATER ON 1.2
      AND     X190F  ; EM.STOP NO1.2
      AND     X1900  ; INV.CONVEYOR BEFORE HEATER
      ANI     B55B  ; GP.CONV OUT B/F HEATER OFF 1.2
      OUT     Y1920  ; INV.CONVEYOR BEFORE HEATER
      OUT     B65A  ; GP.LAMP CON. OUT B/F HEATER 1.2
25    LD      X1905  ; CS.MANUAL/AUTO 1.2
      AND     M1231  ; CONVEYOR FEED OUT2 (BF.HEATER)
      OR      B55C  ; GP.CONVEYOR HEATER NO.1.2 ON
      OR      B555  ; GP.CONV OUT BEFORE HEATER ON 1.2
      ANI     B55D  ; GP.CONVEYOR HEATER NO.1.2 OFF
      AND     X1901  ; INV.CONVEYOR HEATER
      OUT     Y1921  ; INV.CONVEYOR HEATER
      OUT     B65C  ; GP.LAMP CONV. HEATER 1.2
33    LD      B552  ; GP.BLOWER HEATER ON NO.1.2
      SET     M502  ; GP.BLOWER HEATER ON
35    LD      B553  ; GP.BLOWER HEATER ON NO.1.2
      OR      B540  ; AUTO MODE TO POWDER
      RST     M502  ; GP.BLOWER HEATER ON
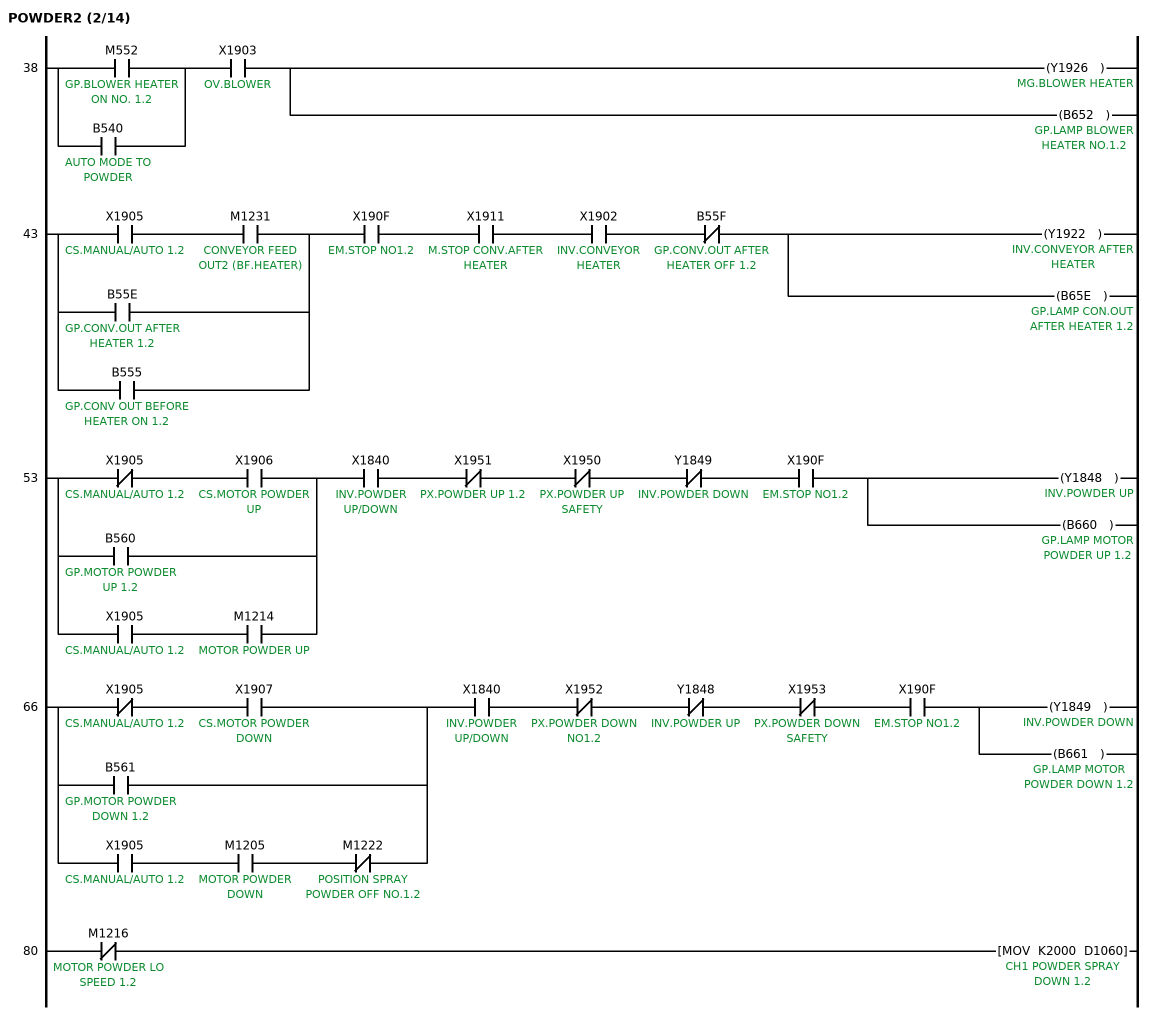
38    LD      M552  ; GP.BLOWER HEATER ON NO. 1.2
      OR      B540  ; AUTO MODE TO POWDER
      AND     X1903  ; OV.BLOWER
      OUT     Y1926  ; MG.BLOWER HEATER
      OUT     B652  ; GP.LAMP BLOWER HEATER NO.1.2
43    LD      X1905  ; CS.MANUAL/AUTO 1.2
      AND     M1231  ; CONVEYOR FEED OUT2 (BF.HEATER)
      OR      B55E  ; GP.CONV.OUT AFTER HEATER 1.2
      OR      B555  ; GP.CONV OUT BEFORE HEATER ON 1.2
      AND     X190F  ; EM.STOP NO1.2
      AND     X1911  ; M.STOP CONV.AFTER HEATER
      AND     X1902  ; INV.CONVEYOR HEATER
      ANI     B55F  ; GP.CONV.OUT AFTER HEATER OFF 1.2
      OUT     Y1922  ; INV.CONVEYOR AFTER HEATER
      OUT     B65E  ; GP.LAMP CON.OUT AFTER HEATER 1.2
53    LDI     X1905  ; CS.MANUAL/AUTO 1.2
      AND     X1906  ; CS.MOTOR POWDER UP
      OR      B560  ; GP.MOTOR POWDER UP 1.2
      LD      X1905  ; CS.MANUAL/AUTO 1.2
      AND     M1214  ; MOTOR POWDER UP
      ORB
      AND     X1840  ; INV.POWDER UP/DOWN
      ANI     X1951  ; PX.POWDER UP 1.2
      ANI     X1950  ; PX.POWDER UP SAFETY
      ANI     Y1849  ; INV.POWDER DOWN
      AND     X190F  ; EM.STOP NO1.2
      OUT     Y1848  ; INV.POWDER UP
      OUT     B660  ; GP.LAMP MOTOR POWDER UP 1.2
66    LDI     X1905  ; CS.MANUAL/AUTO 1.2
      AND     X1907  ; CS.MOTOR POWDER DOWN
      OR      B561  ; GP.MOTOR POWDER DOWN 1.2
      LD      X1905  ; CS.MANUAL/AUTO 1.2
      AND     M1205  ; MOTOR POWDER DOWN
      ANI     M1222  ; POSITION SPRAY POWDER OFF NO.1.2
      ORB
      AND     X1840  ; INV.POWDER UP/DOWN
      ANI     X1952  ; PX.POWDER DOWN NO1.2
      ANI     Y1848  ; INV.POWDER UP
      ANI     X1953  ; PX.POWDER DOWN SAFETY
      AND     X190F  ; EM.STOP NO1.2
      OUT     Y1849  ; INV.POWDER DOWN
      OUT     B661  ; GP.LAMP MOTOR POWDER DOWN 1.2
80    LDI     M1216  ; MOTOR POWDER LO SPEED 1.2
      MOV     K2000 D1060  ; CH1 POWDER SPRAY DOWN 1.2
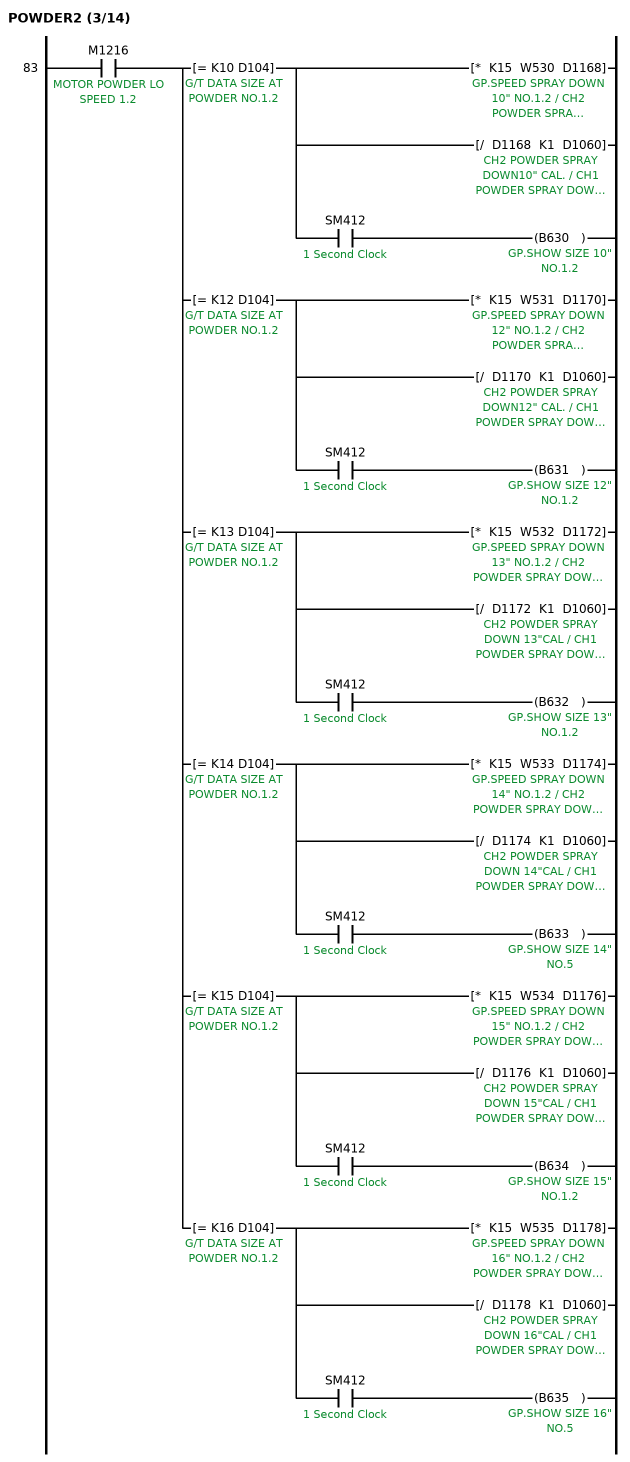
83    LD      M1216  ; MOTOR POWDER LO SPEED 1.2
      MPS
      AND=    K10 D104  ; G/T DATA SIZE AT POWDER NO.1.2
      *       K15 W530 D1168  ; GP.SPEED SPRAY DOWN 10" NO.1.2 / CH2 POWDER SPRAY DOWN10" CAL.
      /       D1168 K1 D1060
      AND     SM412  ; 1 Second Clock
      OUT     B630  ; GP.SHOW SIZE 10" NO.1.2
      MRD
      AND=    K12 D104  ; G/T DATA SIZE AT POWDER NO.1.2
      *       K15 W531 D1170  ; GP.SPEED SPRAY DOWN 12" NO.1.2 / CH2 POWDER SPRAY DOWN12" CAL.
      /       D1170 K1 D1060
      AND     SM412  ; 1 Second Clock
      OUT     B631  ; GP.SHOW SIZE 12" NO.1.2
      MRD
      AND=    K13 D104  ; G/T DATA SIZE AT POWDER NO.1.2
      *       K15 W532 D1172  ; GP.SPEED SPRAY DOWN 13" NO.1.2 / CH2 POWDER SPRAY DOWN 13"CAL
      /       D1172 K1 D1060
      AND     SM412  ; 1 Second Clock
      OUT     B632  ; GP.SHOW SIZE 13" NO.1.2
      MRD
      AND=    K14 D104  ; G/T DATA SIZE AT POWDER NO.1.2
      *       K15 W533 D1174  ; GP.SPEED SPRAY DOWN 14" NO.1.2 / CH2 POWDER SPRAY DOWN 14"CAL
      /       D1174 K1 D1060
      AND     SM412  ; 1 Second Clock
      OUT     B633  ; GP.SHOW SIZE 14" NO.5
      MRD
      AND=    K15 D104  ; G/T DATA SIZE AT POWDER NO.1.2
      *       K15 W534 D1176  ; GP.SPEED SPRAY DOWN 15" NO.1.2 / CH2 POWDER SPRAY DOWN 15"CAL
      /       D1176 K1 D1060
      AND     SM412  ; 1 Second Clock
      OUT     B634  ; GP.SHOW SIZE 15" NO.1.2
      MPP
      AND=    K16 D104  ; G/T DATA SIZE AT POWDER NO.1.2
      *       K15 W535 D1178  ; GP.SPEED SPRAY DOWN 16" NO.1.2 / CH2 POWDER SPRAY DOWN 16"CAL
      /       D1178 K1 D1060
      AND     SM412  ; 1 Second Clock
      OUT     B635  ; GP.SHOW SIZE 16" NO.5
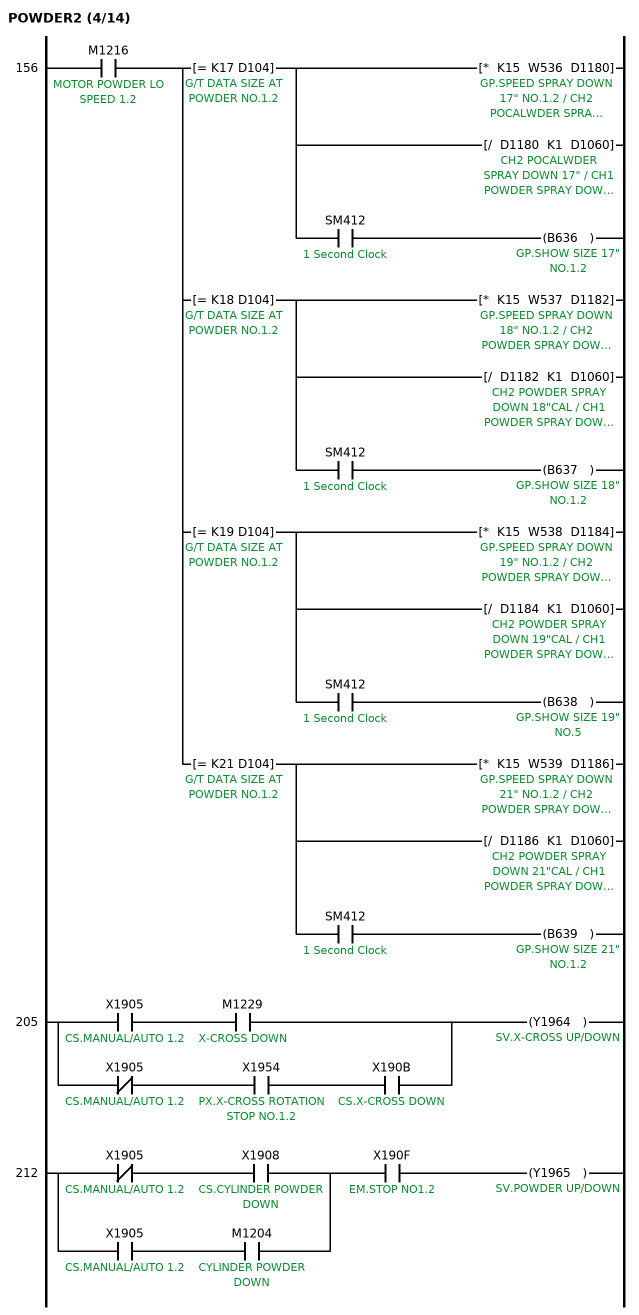
156   LD      M1216  ; MOTOR POWDER LO SPEED 1.2
      MPS
      AND=    K17 D104  ; G/T DATA SIZE AT POWDER NO.1.2
      *       K15 W536 D1180  ; GP.SPEED SPRAY DOWN 17" NO.1.2 / CH2 POCALWDER SPRAY DOWN 17"
      /       D1180 K1 D1060
      AND     SM412  ; 1 Second Clock
      OUT     B636  ; GP.SHOW SIZE 17" NO.1.2
      MRD
      AND=    K18 D104  ; G/T DATA SIZE AT POWDER NO.1.2
      *       K15 W537 D1182  ; GP.SPEED SPRAY DOWN 18" NO.1.2 / CH2 POWDER SPRAY DOWN 18"CAL
      /       D1182 K1 D1060
      AND     SM412  ; 1 Second Clock
      OUT     B637  ; GP.SHOW SIZE 18" NO.1.2
      MRD
      AND=    K19 D104  ; G/T DATA SIZE AT POWDER NO.1.2
      *       K15 W538 D1184  ; GP.SPEED SPRAY DOWN 19" NO.1.2 / CH2 POWDER SPRAY DOWN 19"CAL
      /       D1184 K1 D1060
      AND     SM412  ; 1 Second Clock
      OUT     B638  ; GP.SHOW SIZE 19" NO.5
      MPP
      AND=    K21 D104  ; G/T DATA SIZE AT POWDER NO.1.2
      *       K15 W539 D1186  ; GP.SPEED SPRAY DOWN 21" NO.1.2 / CH2 POWDER SPRAY DOWN 21"CAL
      /       D1186 K1 D1060
      AND     SM412  ; 1 Second Clock
      OUT     B639  ; GP.SHOW SIZE 21" NO.1.2
205   LD      X1905  ; CS.MANUAL/AUTO 1.2
      AND     M1229  ; X-CROSS DOWN
      LDI     X1905  ; CS.MANUAL/AUTO 1.2
      AND     X1954  ; PX.X-CROSS ROTATION STOP NO.1.2
      AND     X190B  ; CS.X-CROSS DOWN
      ORB
      OUT     Y1964  ; SV.X-CROSS UP/DOWN
212   LDI     X1905  ; CS.MANUAL/AUTO 1.2
      AND     X1908  ; CS.CYLINDER POWDER DOWN
      LD      X1905  ; CS.MANUAL/AUTO 1.2
      AND     M1204  ; CYLINDER POWDER DOWN
      ORB
      AND     X190F  ; EM.STOP NO1.2
      OUT     Y1965  ; SV.POWDER UP/DOWN
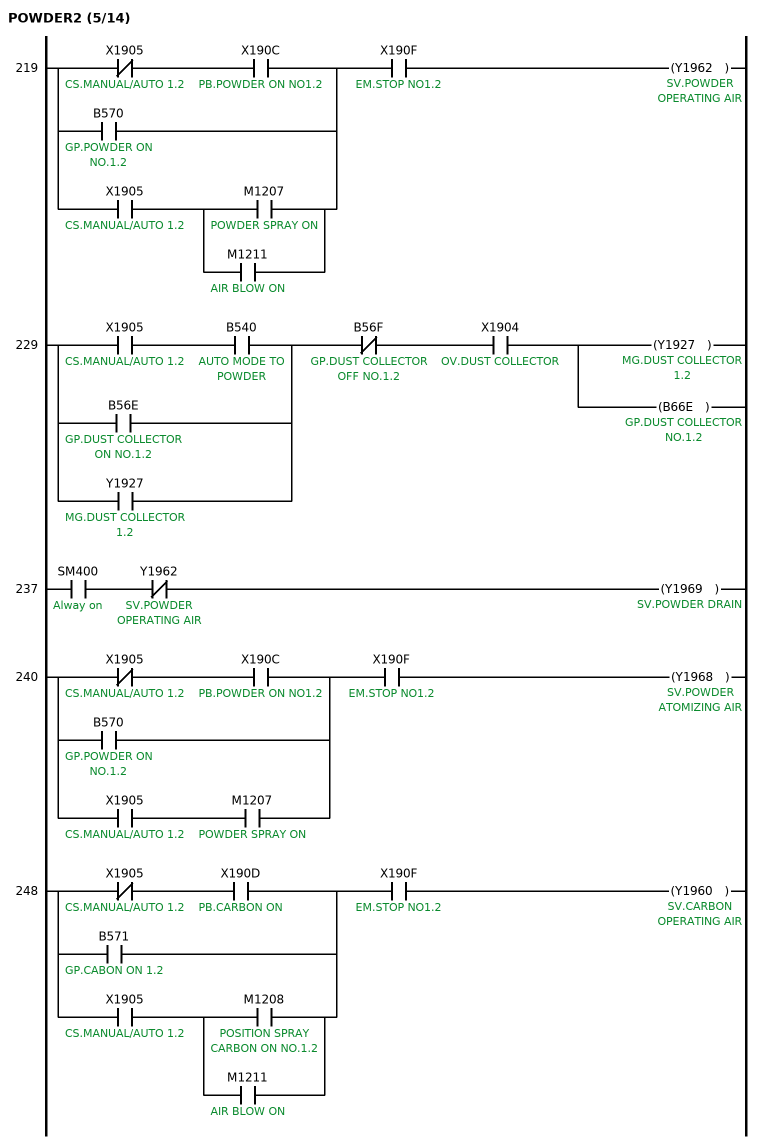
219   LDI     X1905  ; CS.MANUAL/AUTO 1.2
      AND     X190C  ; PB.POWDER ON NO1.2
      OR      B570  ; GP.POWDER ON NO.1.2
      LD      X1905  ; CS.MANUAL/AUTO 1.2
      LD      M1207  ; POWDER SPRAY ON
      OR      M1211  ; AIR BLOW ON
      ANB
      ORB
      AND     X190F  ; EM.STOP NO1.2
      OUT     Y1962  ; SV.POWDER OPERATING AIR
229   LD      X1905  ; CS.MANUAL/AUTO 1.2
      AND     B540  ; AUTO MODE TO POWDER
      OR      B56E  ; GP.DUST COLLECTOR ON NO.1.2
      OR      Y1927  ; MG.DUST COLLECTOR 1.2
      ANI     B56F  ; GP.DUST COLLECTOR OFF NO.1.2
      AND     X1904  ; OV.DUST COLLECTOR
      OUT     Y1927  ; MG.DUST COLLECTOR 1.2
      OUT     B66E  ; GP.DUST COLLECTOR NO.1.2
237   LD      SM400  ; Alway on
      ANI     Y1962  ; SV.POWDER OPERATING AIR
      OUT     Y1969  ; SV.POWDER DRAIN
240   LDI     X1905  ; CS.MANUAL/AUTO 1.2
      AND     X190C  ; PB.POWDER ON NO1.2
      OR      B570  ; GP.POWDER ON NO.1.2
      LD      X1905  ; CS.MANUAL/AUTO 1.2
      AND     M1207  ; POWDER SPRAY ON
      ORB
      AND     X190F  ; EM.STOP NO1.2
      OUT     Y1968  ; SV.POWDER ATOMIZING AIR
248   LDI     X1905  ; CS.MANUAL/AUTO 1.2
      AND     X190D  ; PB.CARBON ON
      OR      B571  ; GP.CABON ON 1.2
      LD      X1905  ; CS.MANUAL/AUTO 1.2
      LD      M1208  ; POSITION SPRAY CARBON ON NO.1.2
      OR      M1211  ; AIR BLOW ON
      ANB
      ORB
      AND     X190F  ; EM.STOP NO1.2
      OUT     Y1960  ; SV.CARBON OPERATING AIR
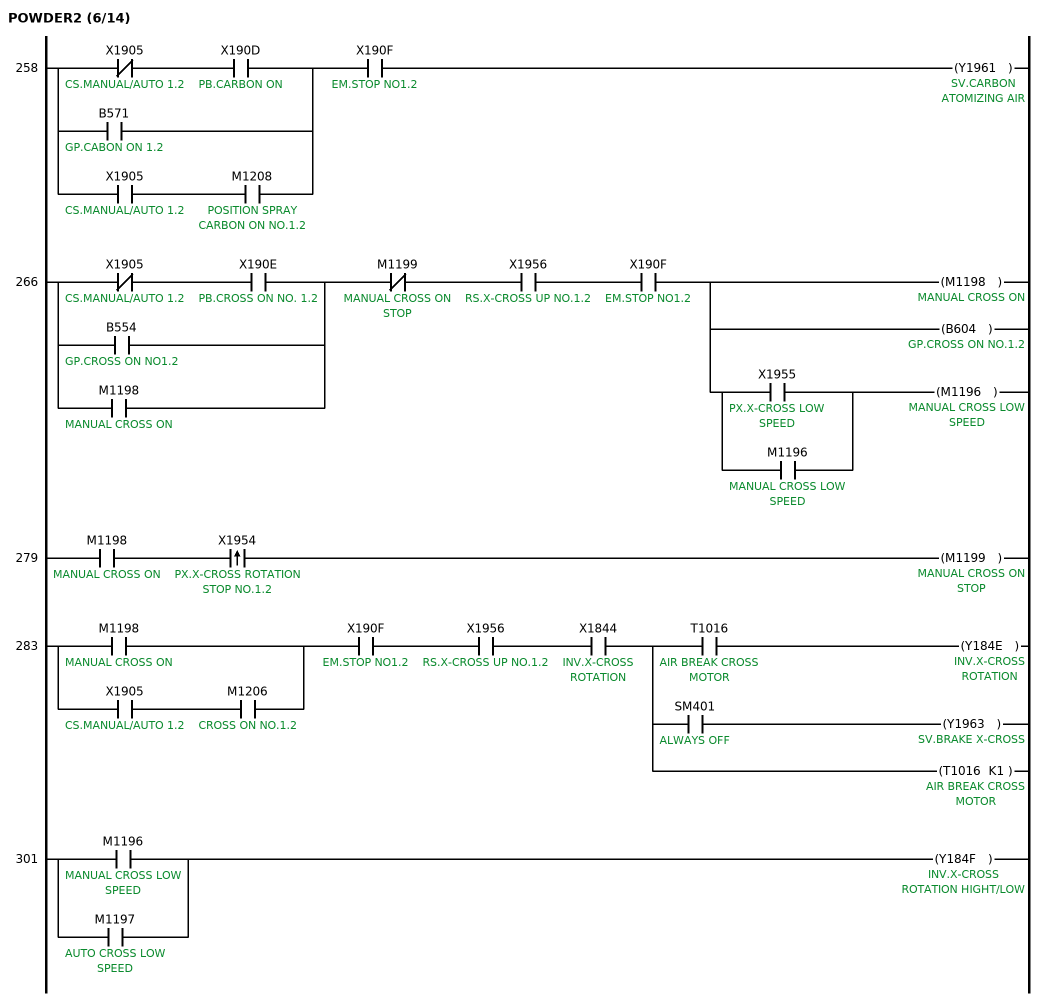
258   LDI     X1905  ; CS.MANUAL/AUTO 1.2
      AND     X190D  ; PB.CARBON ON
      OR      B571  ; GP.CABON ON 1.2
      LD      X1905  ; CS.MANUAL/AUTO 1.2
      AND     M1208  ; POSITION SPRAY CARBON ON NO.1.2
      ORB
      AND     X190F  ; EM.STOP NO1.2
      OUT     Y1961  ; SV.CARBON ATOMIZING AIR
266   LDI     X1905  ; CS.MANUAL/AUTO 1.2
      AND     X190E  ; PB.CROSS ON NO. 1.2
      OR      B554  ; GP.CROSS ON NO1.2
      OR      M1198  ; MANUAL CROSS ON
      ANI     M1199  ; MANUAL CROSS ON STOP
      AND     X1956  ; RS.X-CROSS UP NO.1.2
      AND     X190F  ; EM.STOP NO1.2
      OUT     M1198  ; MANUAL CROSS ON
      OUT     B604  ; GP.CROSS ON NO.1.2
      LD      X1955  ; PX.X-CROSS LOW SPEED
      OR      M1196  ; MANUAL CROSS LOW SPEED
      ANB
      OUT     M1196  ; MANUAL CROSS LOW SPEED
279   LD      M1198  ; MANUAL CROSS ON
      ANDP    X1954  ; PX.X-CROSS ROTATION STOP NO.1.2
      OUT     M1199  ; MANUAL CROSS ON STOP
283   LD      M1198  ; MANUAL CROSS ON
      LD      X1905  ; CS.MANUAL/AUTO 1.2
      AND     M1206  ; CROSS ON NO.1.2
      ORB
      AND     X190F  ; EM.STOP NO1.2
      AND     X1956  ; RS.X-CROSS UP NO.1.2
      AND     X1844  ; INV.X-CROSS ROTATION
      MPS
      AND     T1016  ; AIR BREAK CROSS MOTOR
      OUT     Y184E  ; INV.X-CROSS ROTATION
      MRD
      AND     SM401  ; ALWAYS OFF
      OUT     Y1963  ; SV.BRAKE X-CROSS
      MPP
      OUT     T1016 K1  ; AIR BREAK CROSS MOTOR
301   LD      M1196  ; MANUAL CROSS LOW SPEED
      OR      M1197  ; AUTO CROSS LOW SPEED
      OUT     Y184F  ; INV.X-CROSS ROTATION HIGHT/LOW
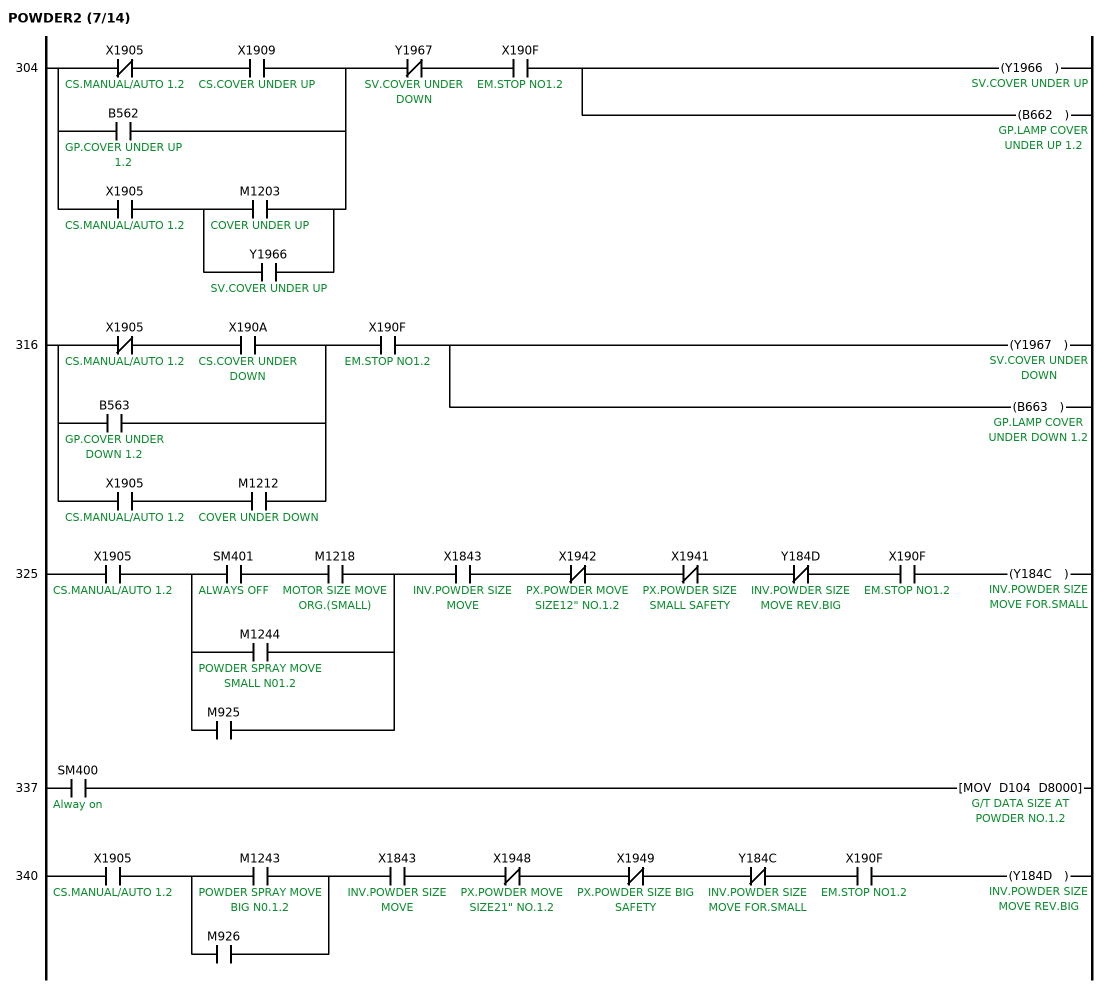
304   LDI     X1905  ; CS.MANUAL/AUTO 1.2
      AND     X1909  ; CS.COVER UNDER UP
      OR      B562  ; GP.COVER UNDER UP 1.2
      LD      X1905  ; CS.MANUAL/AUTO 1.2
      LD      M1203  ; COVER UNDER UP
      OR      Y1966  ; SV.COVER UNDER UP
      ANB
      ORB
      ANI     Y1967  ; SV.COVER UNDER DOWN
      AND     X190F  ; EM.STOP NO1.2
      OUT     Y1966  ; SV.COVER UNDER UP
      OUT     B662  ; GP.LAMP COVER UNDER UP 1.2
316   LDI     X1905  ; CS.MANUAL/AUTO 1.2
      AND     X190A  ; CS.COVER UNDER DOWN
      OR      B563  ; GP.COVER UNDER DOWN 1.2
      LD      X1905  ; CS.MANUAL/AUTO 1.2
      AND     M1212  ; COVER UNDER DOWN
      ORB
      AND     X190F  ; EM.STOP NO1.2
      OUT     Y1967  ; SV.COVER UNDER DOWN
      OUT     B663  ; GP.LAMP COVER UNDER DOWN 1.2
325   LD      X1905  ; CS.MANUAL/AUTO 1.2
      LD      SM401  ; ALWAYS OFF
      AND     M1218  ; MOTOR SIZE MOVE ORG.(SMALL)
      OR      M1244  ; POWDER SPRAY MOVE SMALL N01.2
      OR      M925
      ANB
      AND     X1843  ; INV.POWDER SIZE MOVE
      ANI     X1942  ; PX.POWDER MOVE SIZE12" NO.1.2
      ANI     X1941  ; PX.POWDER SIZE SMALL SAFETY
      ANI     Y184D  ; INV.POWDER SIZE MOVE REV.BIG
      AND     X190F  ; EM.STOP NO1.2
      OUT     Y184C  ; INV.POWDER SIZE MOVE FOR.SMALL
337   LD      SM400  ; Alway on
      MOV     D104 D8000
340   LD      X1905  ; CS.MANUAL/AUTO 1.2
      LD      M1243  ; POWDER SPRAY MOVE  BIG N0.1.2
      OR      M926
      ANB
      AND     X1843  ; INV.POWDER SIZE MOVE
      ANI     X1948  ; PX.POWDER MOVE SIZE21" NO.1.2
      ANI     X1949  ; PX.POWDER SIZE BIG SAFETY
      ANI     Y184C  ; INV.POWDER SIZE MOVE FOR.SMALL
      AND     X190F  ; EM.STOP NO1.2
      OUT     Y184D  ; INV.POWDER SIZE MOVE REV.BIG
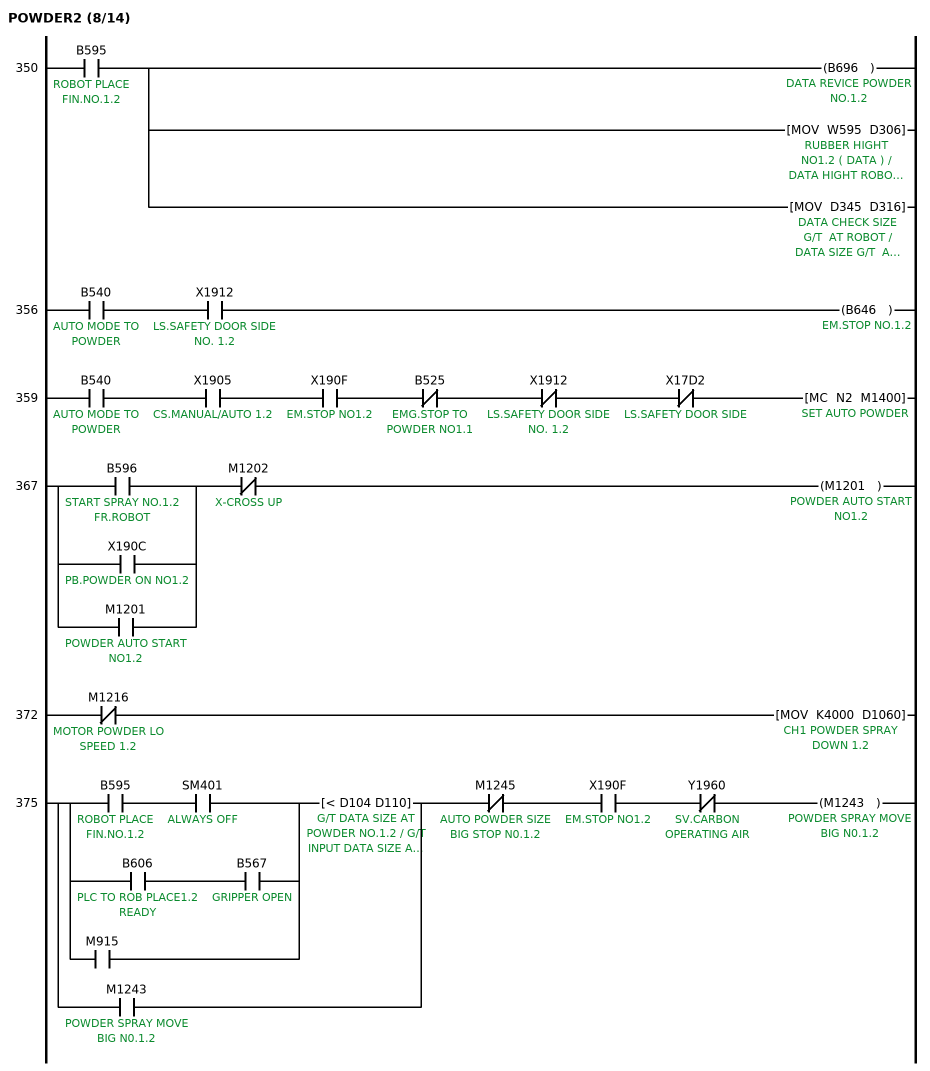
350   LD      B595  ; ROBOT PLACE FIN.NO.1.2
      OUT     B696  ; DATA REVICE POWDER NO.1.2
      MOV     W595 D306  ; RUBBER HIGHT NO1.2 ( DATA ) / DATA HIGHT ROBOT TO N0.1.2
      MOV     D345 D316  ; DATA CHECK SIZE G/T  AT ROBOT / DATA SIZE G/T  AT ROBOT NO.1.2
356   LD      B540  ; AUTO MODE TO POWDER
      AND     X1912  ; LS.SAFETY DOOR SIDE NO. 1.2
      OUT     B646  ; EM.STOP NO.1.2
359   LD      B540  ; AUTO MODE TO POWDER
      AND     X1905  ; CS.MANUAL/AUTO 1.2
      AND     X190F  ; EM.STOP NO1.2
      ANI     B525  ; EMG.STOP TO POWDER NO1.1
      ANI     X1912  ; LS.SAFETY DOOR SIDE NO. 1.2
      ANI     X17D2  ; LS.SAFETY DOOR SIDE
      MC      N2 M1400  ; SET AUTO POWDER
367   LD      B596  ; START SPRAY NO.1.2 FR.ROBOT
      OR      X190C  ; PB.POWDER ON NO1.2
      OR      M1201  ; POWDER AUTO START NO1.2
      ANI     M1202  ; X-CROSS UP
      OUT     M1201  ; POWDER AUTO START NO1.2
372   LDI     M1216  ; MOTOR POWDER LO SPEED 1.2
      MOV     K4000 D1060
375   LD      B595  ; ROBOT PLACE FIN.NO.1.2
      AND     SM401  ; ALWAYS OFF
      LD      B606  ; PLC TO ROB PLACE1.2 READY
      AND     B567  ; GRIPPER OPEN
      ORB
      OR      M915
      AND<    D104 D110  ; G/T DATA SIZE AT POWDER NO.1.2 / G/T INPUT DATA SIZE AT ROBOT
      OR      M1243  ; POWDER SPRAY MOVE  BIG N0.1.2
      ANI     M1245  ; AUTO POWDER SIZE BIG STOP N0.1.2
      AND     X190F  ; EM.STOP NO1.2
      ANI     Y1960  ; SV.CARBON OPERATING AIR
      OUT     M1243  ; POWDER SPRAY MOVE  BIG N0.1.2
